KUKA KRL program: EPS_2_25252_SD1A_A_20250910061717.src

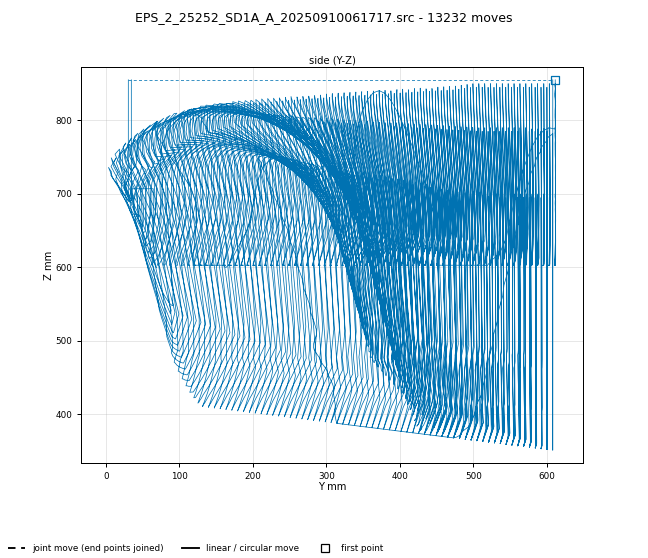
[picture p0: tool path of EPS_2_25252_SD1A_A_20250910061717.src, 13232 of 13234 moves have a stored position in this frame; points joined in program order, loops and branches not executed]
&ACCESS RVP
&REL 4
&COMMENT QRS 19112012
&PARAM EDITMASK = *
DEF PART()
EXT BAS (BAS_COMMAND :IN,REAL :IN )
INT I
BAS (#INITMOV,0 )

;KUKA QRS Post kuka4.cps  Date:22-06-2017 !

File_ID=2822

QRS_PRE_INIT()

;Init var - Until changes are made in qrs_pre_init
Outlet_Square_prg=0
Inlet_1_Square_prg=0
Inlet_2_Square_prg=0
Inlet_3_Square_prg=0
Inlet_4_Square_prg=0
Inlet_5_Square_prg=0

Outlet_1={X 0.000, Y 501.250, Z 662.000, B 0.000, E1 0.000 }
Inlet_1={X 0.000, Y 505.750, Z 602.000, B 0.000, E1 90.000 }
Inlet_2={X 0.000, Y 531.500, Z 514.500, B 0.000, E1 270.000 }
Outlet_1_type=366
Inlet_1_type=366
Inlet_2_type=201
;QRS#1=Sidecore dimensions
;QRS#2=375-15" PVC SDR 35
;QRS#3=375-15" PVC SDR 35
;QRS#4=200-8" PVC SDR 35
;QRS#5=
;QRS#6=
;QRS#7=
;QRS#8=
;QRS#9=20Y PSX
;QRS#10=20Y PSX
;QRS#11=12-08 PSX
;QRS#12=
;QRS#13=
;QRS#14=
;QRS#15=
;QRS#16=1220x127x1143 3,75'
;QRS#17=EPS Height
;QRS#18=845
;QRS#19=*
;QRS#20= UPDATED VERSION 22-06-2017
;QRS#21=*
Outlet_Square=0250
Inlet_1_Square=0250
Inlet_2_Square=0100
Inlet_3_Square=0
Inlet_4_Square=0
Inlet_5_Square=0
Mill_Square=1
Outlet_Square_Prg=252
Inlet_1_Square_prg=252
Inlet_2_Square_prg=204

QRS_INIT()

$ADVANCE=5

; T1
PTP {E1 176.989,E2 176.989}
PTP {X 0,Y 611.255,A -85,B 0,C 180,E1 176.989,E2 176.989,E3 0,E4 0,E5 0,E6 0}
QRS_SPEED_INIT()
LIN {X 0,Y 611.255,Z 855,A -85,B 0,C 180,E1 176.989,E2 176.989,E3 0,E4 0,E5 0,E6 0} C_VEL
LIN {X 0,Y 611.255,Z 797.706,A -85,B 0,C 180,E1 176.989,E2 176.989} C_VEL
LIN {X 0,Y 611.255,Z 789.909,A -85,B 0,C 180,E1 176.989,E2 176.989} C_VEL
LIN {X 0,Y 611.338,Z 787.921,A -85,B 0,C 180,E1 177.197,E2 177.197} C_VEL
LIN {X 0,Y 611.834,Z 789.089,A -85,B 0,C 180,E1 178.169,E2 178.169} C_VEL
LIN {X 0,Y 611.558,Z 789.587,A -85,B 0,C 180,E1 178.832,E2 178.832} C_VEL
LIN {X 0,Y 611.055,Z 789.944,A -85,B 0,C 180,E1 179.766,E2 179.766} C_VEL
LIN {X 0,Y 610.786,Z 789.821,A -85,B 0,C 180,E1 180.701,E2 180.701} C_VEL
LIN {X 0,Y 610.813,Z 789.552,A -85,B 0,C 180,E1 181.169,E2 181.169} C_VEL
LIN {X 0,Y 611.351,Z 788.136,A -85,B 0,C 180,E1 182.57,E2 182.57} C_VEL
LIN {X 0,Y 611.881,Z 786.565,A -85,B 0,C 180,E1 183.503,E2 183.503} C_VEL
LIN {X 0,Y 611.302,Z 783.918,A -85,B 0,C 180,E1 184.677,E2 184.677} C_VEL
LIN {X 0,Y 611.043,Z 782.348,A -85,B 0,C 180,E1 185.266,E2 185.266} C_VEL
LIN {X 0,Y 610.913,Z 779.545,A -85,B 0,C 180,E1 186.148,E2 186.148} C_VEL
LIN {X 0,Y 611.141,Z 776.265,A -85,B 0,C 180,E1 187.027,E2 187.027} C_VEL
LIN {X 0,Y 611.585,Z 772.483,A -85,B 0,C 180,E1 187.905,E2 187.905} C_VEL
LIN {X 0,Y 611.869,Z 769.622,A -85,B 0,C 180,E1 188.491,E2 188.491} C_VEL
LIN {X 0,Y 611.527,Z 764.94,A -85,B 0,C 180,E1 189.382,E2 189.382} C_VEL
LIN {X 0,Y 611.202,Z 759.672,A -85,B 0,C 180,E1 190.276,E2 190.276} C_VEL
LIN {X 0,Y 611.223,Z 752.664,A -85,B 0,C 180,E1 191.317,E2 191.317} C_VEL
LIN {X 0,Y 611.512,Z 747.064,A -85,B 0,C 180,E1 192.056,E2 192.056} C_VEL
LIN {X 0,Y 611.803,Z 740.897,A -85,B 0,C 180,E1 192.797,E2 192.797} C_VEL
LIN {X 0,Y 611.777,Z 735.91,A -85,B 0,C 180,E1 193.359,E2 193.359} C_VEL
LIN {X 0,Y 611.519,Z 727.994,A -85,B 0,C 180,E1 194.172,E2 194.172} C_VEL
LIN {X 0,Y 611.4,Z 721.632,A -85,B 0,C 180,E1 194.769,E2 194.769} C_VEL
LIN {X 0,Y 611.46,Z 714.699,A -85,B 0,C 180,E1 195.363,E2 195.363} C_VEL
LIN {X 0,Y 611.677,Z 706.786,A -85,B 0,C 180,E1 195.978,E2 195.978} C_VEL
LIN {X 0,Y 611.783,Z 698.644,A -85,B 0,C 180,E1 196.557,E2 196.557} C_VEL
LIN {X 0,Y 611.811,Z 690.326,A -85,B 0,C 180,E1 197.094,E2 197.094} C_VEL
LIN {X 0,Y 611.741,Z 682.443,A -85,B 0,C 180,E1 197.56,E2 197.56} C_VEL
LIN {X 0,Y 611.722,Z 675.291,A -85,B 0,C 180,E1 197.945,E2 197.945} C_VEL
LIN {X 0,Y 611.776,Z 665.714,A -85,B 0,C 180,E1 198.404,E2 198.404} C_VEL
LIN {X 0,Y 611.781,Z 656.669,A -85,B 0,C 180,E1 198.789,E2 198.789} C_VEL
LIN {X 0,Y 611.797,Z 648.504,A -85,B 0,C 180,E1 199.097,E2 199.097} C_VEL
LIN {X 0,Y 611.848,Z 637.724,A -85,B 0,C 180,E1 199.443,E2 199.443} C_VEL
LIN {X 0,Y 611.821,Z 629.276,A -85,B 0,C 180,E1 199.676,E2 199.676} C_VEL
LIN {X 0,Y 611.827,Z 618.943,A -85,B 0,C 180,E1 199.908,E2 199.908} C_VEL
LIN {X 0,Y 611.776,Z 610.345,A -85,B 0,C 180,E1 200.065,E2 200.065} C_VEL
LIN {X 0,Y 611.596,Z 602.81,A -85,B 0,C 180,E1 200.188,E2 200.188} C_VEL
LIN {X 0,Y 611.78,Z 602.81,A -85,B 0,C 180,E1 200.26,E2 200.26} C_VEL
LIN {X 0,Y 611.752,Z 602.81,A -85,B 0,C 180,E1 207.938,E2 207.938} C_VEL
LIN {X 0,Y 610.419,Z 602.81,A -85,B 0,C 180,E1 210.688,E2 210.688} C_VEL
LIN {X 0,Y 611.718,Z 602.81,A -85,B 0,C 180,E1 216.211,E2 216.211} C_VEL
LIN {X 0,Y 611.159,Z 602.81,A -85,B 0,C 180,E1 217.326,E2 217.326} C_VEL
LIN {X 0,Y 610.678,Z 602.81,A -85,B 0,C 180,E1 222.329,E2 222.329} C_VEL
LIN {X 0,Y 611.693,Z 602.81,A -85,B 0,C 180,E1 224.519,E2 224.519} C_VEL
LIN {X 0,Y 611.666,Z 602.81,A -85,B 0,C 180,E1 232.612,E2 232.612} C_VEL
LIN {X 0,Y 611.151,Z 602.81,A -85,B 0,C 180,E1 233.75,E2 233.75} C_VEL
LIN {X 0,Y 611.656,Z 602.81,A -85,B 0,C 180,E1 241.169,E2 241.169} C_VEL
LIN {X 0,Y 611.476,Z 602.81,A -85,B 0,C 180,E1 242.049,E2 242.049} C_VEL
LIN {X 0,Y 611.803,Z 602.81,A -85,B 0,C 180,E1 248.625,E2 248.625} C_VEL
LIN {X 0,Y 610.997,Z 602.81,A -85,B 0,C 180,E1 248.983,E2 248.983} C_VEL
LIN {X 0,Y 610.769,Z 602.853,A -85,B 0,C 180,E1 249.009,E2 249.009} C_VEL
LIN {X 0,Y 611.62,Z 640.893,A -85,B 0,C 180,E1 249.507,E2 249.507} C_VEL
LIN {X 0,Y 611.825,Z 668.068,A -85,B 0,C 180,E1 249.859,E2 249.859} C_VEL
LIN {X 0,Y 611.844,Z 677.232,A -85,B 0,C 180,E1 250.014,E2 250.014} C_VEL
LIN {X 0,Y 611.82,Z 686.284,A -85,B 0,C 180,E1 250.208,E2 250.208} C_VEL
LIN {X 0,Y 611.674,Z 695.239,A -85,B 0,C 180,E1 250.435,E2 250.435} C_VEL
LIN {X 0,Y 611.805,Z 704.1,A -85,B 0,C 180,E1 250.71,E2 250.71} C_VEL
LIN {X 0,Y 611.808,Z 711.864,A -85,B 0,C 180,E1 250.981,E2 250.981} C_VEL
LIN {X 0,Y 611.808,Z 721.496,A -85,B 0,C 180,E1 251.366,E2 251.366} C_VEL
LIN {X 0,Y 611.827,Z 729.998,A -85,B 0,C 180,E1 251.751,E2 251.751} C_VEL
LIN {X 0,Y 611.756,Z 739.053,A -85,B 0,C 180,E1 252.209,E2 252.209} C_VEL
LIN {X 0,Y 611.731,Z 748.469,A -85,B 0,C 180,E1 252.745,E2 252.745} C_VEL
LIN {X 0,Y 611.565,Z 756.855,A -85,B 0,C 180,E1 253.272,E2 253.272} C_VEL
LIN {X 0,Y 611.462,Z 763.316,A -85,B 0,C 180,E1 253.715,E2 253.715} C_VEL
LIN {X 0,Y 611.523,Z 770.776,A -85,B 0,C 180,E1 254.277,E2 254.277} C_VEL
LIN {X 0,Y 611.733,Z 778.696,A -85,B 0,C 180,E1 254.937,E2 254.937} C_VEL
LIN {X 0,Y 611.827,Z 785.197,A -85,B 0,C 180,E1 255.523,E2 255.523} C_VEL
LIN {X 0,Y 611.641,Z 792.111,A -85,B 0,C 180,E1 256.198,E2 256.198} C_VEL
LIN {X 0,Y 611.381,Z 798.097,A -85,B 0,C 180,E1 256.831,E2 256.831} C_VEL
LIN {X 0,Y 611.254,Z 803.807,A -85,B 0,C 180,E1 257.49,E2 257.49} C_VEL
LIN {X 0,Y 611.36,Z 809.701,A -85,B 0,C 180,E1 258.239,E2 258.239} C_VEL
LIN {X 0,Y 611.556,Z 814.069,A -85,B 0,C 180,E1 258.838,E2 258.838} C_VEL
LIN {X 0,Y 611.862,Z 819.944,A -85,B 0,C 180,E1 259.735,E2 259.735} C_VEL
LIN {X 0,Y 611.48,Z 825.185,A -85,B 0,C 180,E1 260.617,E2 260.617} C_VEL
LIN {X 0,Y 611.206,Z 828.398,A -85,B 0,C 180,E1 261.204,E2 261.204} C_VEL
LIN {X 0,Y 611.051,Z 832.684,A -85,B 0,C 180,E1 262.088,E2 262.088} C_VEL
LIN {X 0,Y 611.215,Z 836.436,A -85,B 0,C 180,E1 262.974,E2 262.974} C_VEL
LIN {X 0,Y 611.602,Z 839.681,A -85,B 0,C 180,E1 263.859,E2 263.859} C_VEL
LIN {X 0,Y 611.753,Z 840.616,A -85,B 0,C 180,E1 264.154,E2 264.154} C_VEL
LIN {X 0,Y 611.721,Z 842.453,A -85,B 0,C 180,E1 264.74,E2 264.74} C_VEL
LIN {X 0,Y 611.158,Z 845.43,A -85,B 0,C 180,E1 265.908,E2 265.908} C_VEL
LIN {X 0,Y 610.966,Z 846.682,A -85,B 0,C 180,E1 266.492,E2 266.492} C_VEL
LIN {X 0,Y 611.091,Z 848.544,A -85,B 0,C 180,E1 267.72,E2 267.72} C_VEL
LIN {X 0,Y 611.598,Z 849.552,A -85,B 0,C 180,E1 268.833,E2 268.833} C_VEL
LIN {X 0,Y 611.713,Z 849.903,A -85,B 0,C 180,E1 269.767,E2 269.767} C_VEL
LIN {X 0,Y 611.245,Z 849.816,A -85,B 0,C 180,E1 270.701,E2 270.701} C_VEL
LIN {X 0,Y 610.955,Z 848.959,A -85,B 0,C 180,E1 271.933,E2 271.933} C_VEL
LIN {X 0,Y 611.441,Z 846.667,A -85,B 0,C 180,E1 273.505,E2 273.505} C_VEL
LIN {X 0,Y 611.736,Z 845.409,A -85,B 0,C 180,E1 274.088,E2 274.088} C_VEL
LIN {X 0,Y 611.745,Z 844.023,A -85,B 0,C 180,E1 274.674,E2 274.674} C_VEL
LIN {X 0,Y 611.452,Z 842.462,A -85,B 0,C 180,E1 275.262,E2 275.262} C_VEL
LIN {X 0,Y 611.033,Z 839.69,A -85,B 0,C 180,E1 276.146,E2 276.146} C_VEL
LIN {X 0,Y 610.903,Z 836.436,A -85,B 0,C 180,E1 277.03,E2 277.03} C_VEL
LIN {X 0,Y 611.133,Z 832.684,A -85,B 0,C 180,E1 277.911,E2 277.911} C_VEL
LIN {X 0,Y 611.587,Z 828.398,A -85,B 0,C 180,E1 278.79,E2 278.79} C_VEL
LIN {X 0,Y 611.871,Z 825.185,A -85,B 0,C 180,E1 279.377,E2 279.377} C_VEL
LIN {X 0,Y 611.518,Z 819.944,A -85,B 0,C 180,E1 280.271,E2 280.271} C_VEL
LIN {X 0,Y 611.154,Z 812.996,A -85,B 0,C 180,E1 281.318,E2 281.318} C_VEL
LIN {X 0,Y 611.164,Z 807.427,A -85,B 0,C 180,E1 282.063,E2 282.063} C_VEL
LIN {X 0,Y 611.414,Z 801.293,A -85,B 0,C 180,E1 282.806,E2 282.806} C_VEL
LIN {X 0,Y 611.786,Z 793.803,A -85,B 0,C 180,E1 283.623,E2 283.623} C_VEL
LIN {X 0,Y 611.787,Z 787.856,A -85,B 0,C 180,E1 284.223,E2 284.223} C_VEL
LIN {X 0,Y 611.566,Z 780.74,A -85,B 0,C 180,E1 284.888,E2 284.888} C_VEL
LIN {X 0,Y 611.417,Z 774.124,A -85,B 0,C 180,E1 285.456,E2 285.456} C_VEL
LIN {X 0,Y 611.438,Z 767.139,A -85,B 0,C 180,E1 286.004,E2 286.004} C_VEL
LIN {X 0,Y 611.599,Z 759.502,A -85,B 0,C 180,E1 286.549,E2 286.549} C_VEL
LIN {X 0,Y 611.777,Z 751.324,A -85,B 0,C 180,E1 287.079,E2 287.079} C_VEL
LIN {X 0,Y 611.815,Z 743.302,A -85,B 0,C 180,E1 287.555,E2 287.555} C_VEL
LIN {X 0,Y 611.798,Z 734.646,A -85,B 0,C 180,E1 288.02,E2 288.02} C_VEL
LIN {X 0,Y 611.708,Z 726.729,A -85,B 0,C 180,E1 288.407,E2 288.407} C_VEL
LIN {X 0,Y 611.712,Z 717.825,A -85,B 0,C 180,E1 288.791,E2 288.791} C_VEL
LIN {X 0,Y 611.801,Z 707.539,A -85,B 0,C 180,E1 289.174,E2 289.174} C_VEL
LIN {X 0,Y 611.768,Z 697.93,A -85,B 0,C 180,E1 289.484,E2 289.484} C_VEL
LIN {X 0,Y 611.774,Z 691.134,A -85,B 0,C 180,E1 289.678,E2 289.678} C_VEL
LIN {X 0,Y 611.852,Z 679.255,A -85,B 0,C 180,E1 289.946,E2 289.946} C_VEL
LIN {X 0,Y 611.842,Z 669.403,A -85,B 0,C 180,E1 290.121,E2 290.121} C_VEL
LIN {X 0,Y 611.69,Z 646.222,A -85,B 0,C 180,E1 290.425,E2 290.425} C_VEL
LIN {X 0,Y 610.919,Z 608.013,A -85,B 0,C 180,E1 290.922,E2 290.922} C_VEL
LIN {X 0,Y 610.821,Z 602.81,A -85,B 0,C 180,E1 290.998,E2 290.998} C_VEL
LIN {X 0,Y 611.662,Z 602.81,A -85,B 0,C 180,E1 291.131,E2 291.131} C_VEL
LIN {X 0,Y 611.599,Z 602.81,A -85,B 0,C 180,E1 291.733,E2 291.733} C_VEL
LIN {X 0,Y 611.815,Z 602.81,A -85,B 0,C 180,E1 297.934,E2 297.934} C_VEL
LIN {X 0,Y 610.481,Z 602.81,A -85,B 0,C 180,E1 300.684,E2 300.684} C_VEL
LIN {X 0,Y 611.803,Z 602.81,A -85,B 0,C 180,E1 306.205,E2 306.205} C_VEL
LIN {X 0,Y 611.22,Z 602.81,A -85,B 0,C 180,E1 307.333,E2 307.333} C_VEL
LIN {X 0,Y 610.732,Z 602.81,A -85,B 0,C 180,E1 312.325,E2 312.325} C_VEL
LIN {X 0,Y 611.759,Z 602.81,A -85,B 0,C 180,E1 314.525,E2 314.525} C_VEL
LIN {X 0,Y 611.719,Z 602.81,A -85,B 0,C 180,E1 322.605,E2 322.605} C_VEL
LIN {X 0,Y 611.181,Z 602.81,A -85,B 0,C 180,E1 323.752,E2 323.752} C_VEL
LIN {X 0,Y 611.606,Z 602.81,A -85,B 0,C 180,E1 331.178,E2 331.178} C_VEL
LIN {X 0,Y 611.391,Z 602.81,A -85,B 0,C 180,E1 332.044,E2 332.044} C_VEL
LIN {X 0,Y 611.822,Z 602.81,A -85,B 0,C 180,E1 339.742,E2 339.742} C_VEL
LIN {X 0,Y 611.83,Z 602.81,A -85,B 0,C 180,E1 347.842,E2 347.842} C_VEL
LIN {X 0,Y 611.645,Z 602.89,A -85,B 0,C 180,E1 348.052,E2 348.052} C_VEL
LIN {X 0,Y 611.831,Z 610.86,A -85,B 0,C 180,E1 348.286,E2 348.286} C_VEL
LIN {X 0,Y 611.839,Z 619.207,A -85,B 0,C 180,E1 348.582,E2 348.582} C_VEL
LIN {X 0,Y 611.857,Z 627.631,A -85,B 0,C 180,E1 348.949,E2 348.949} C_VEL
LIN {X 0,Y 611.843,Z 635.937,A -85,B 0,C 180,E1 349.377,E2 349.377} C_VEL
LIN {X 0,Y 611.694,Z 643.024,A -85,B 0,C 180,E1 349.806,E2 349.806} C_VEL
LIN {X 0,Y 611.601,Z 650.478,A -85,B 0,C 180,E1 350.323,E2 350.323} C_VEL
LIN {X 0,Y 611.746,Z 657.755,A -85,B 0,C 180,E1 350.917,E2 350.917} C_VEL
LIN {X 0,Y 611.865,Z 664.105,A -85,B 0,C 180,E1 351.509,E2 351.509} C_VEL
LIN {X 0,Y 611.633,Z 669.644,A -85,B 0,C 180,E1 352.095,E2 352.095} C_VEL
LIN {X 0,Y 611.278,Z 675.666,A -85,B 0,C 180,E1 352.827,E2 352.827} C_VEL
LIN {X 0,Y 611.236,Z 678.856,A -85,B 0,C 180,E1 353.268,E2 353.268} C_VEL
LIN {X 0,Y 611.382,Z 682.66,A -85,B 0,C 180,E1 353.857,E2 353.857} C_VEL
LIN {X 0,Y 611.667,Z 686.017,A -85,B 0,C 180,E1 354.447,E2 354.447} C_VEL
LIN {X 0,Y 611.88,Z 688.956,A -85,B 0,C 180,E1 355.035,E2 355.035} C_VEL
LIN {X 0,Y 611.599,Z 691.514,A -85,B 0,C 180,E1 355.618,E2 355.618} C_VEL
LIN {X 0,Y 611.128,Z 694.638,A -85,B 0,C 180,E1 356.493,E2 356.493} C_VEL
LIN {X 0,Y 611.022,Z 696.481,A -85,B 0,C 180,E1 357.14,E2 357.14} C_VEL
LIN {X 0,Y 611.323,Z 698.328,A -85,B 0,C 180,E1 358.032,E2 358.032} C_VEL
LIN {X 0,Y 611.76,Z 699.395,A -85,B 0,C 180,E1 358.833,E2 358.833} C_VEL
LIN {X 0,Y 611.815,Z 699.742,A -85,B 0,C 180,E1 359.3,E2 359.3} C_VEL
LIN {X 0,Y 611.316,Z 699.913,A -85,B 0,C 180,E1 360.234,E2 360.234} C_VEL
LIN {X 0,Y 611.123,Z 699.712,A -85,B 0,C 180,E1 360.701,E2 360.701} C_VEL
LIN {X 0,Y 611.058,Z 699.321,A -85,B 0,C 180,E1 361.169,E2 361.169} C_VEL
LIN {X 0,Y 611.126,Z 698.739,A -85,B 0,C 180,E1 361.636,E2 361.636} C_VEL
LIN {X 0,Y 611.568,Z 696.941,A -85,B 0,C 180,E1 362.569,E2 362.569} C_VEL
LIN {X 0,Y 611.798,Z 695.73,A -85,B 0,C 180,E1 363.036,E2 363.036} C_VEL
LIN {X 0,Y 611.681,Z 693.755,A -85,B 0,C 180,E1 363.684,E2 363.684} C_VEL
LIN {X 0,Y 611.326,Z 691.141,A -85,B 0,C 180,E1 364.384,E2 364.384} C_VEL
LIN {X 0,Y 611.126,Z 687.101,A -85,B 0,C 180,E1 365.265,E2 365.265} C_VEL
LIN {X 0,Y 611.288,Z 683.901,A -85,B 0,C 180,E1 365.85,E2 365.85} C_VEL
LIN {X 0,Y 611.771,Z 678.248,A -85,B 0,C 180,E1 366.726,E2 366.726} C_VEL
LIN {X 0,Y 611.814,Z 673.838,A -85,B 0,C 180,E1 367.314,E2 367.314} C_VEL
LIN {X 0,Y 611.505,Z 667.518,A -85,B 0,C 180,E1 368.054,E2 368.054} C_VEL
LIN {X 0,Y 611.396,Z 661.645,A -85,B 0,C 180,E1 368.645,E2 368.645} C_VEL
LIN {X 0,Y 611.567,Z 654.978,A -85,B 0,C 180,E1 369.234,E2 369.234} C_VEL
LIN {X 0,Y 611.802,Z 647.181,A -85,B 0,C 180,E1 369.822,E2 369.822} C_VEL
LIN {X 0,Y 611.792,Z 639.219,A -85,B 0,C 180,E1 370.341,E2 370.341} C_VEL
LIN {X 0,Y 611.673,Z 631.524,A -85,B 0,C 180,E1 370.773,E2 370.773} C_VEL
LIN {X 0,Y 611.667,Z 624.263,A -85,B 0,C 180,E1 371.119,E2 371.119} C_VEL
LIN {X 0,Y 611.771,Z 615.833,A -85,B 0,C 180,E1 371.456,E2 371.456} C_VEL
LIN {X 0,Y 611.596,Z 606.761,A -85,B 0,C 180,E1 371.753,E2 371.753} C_VEL
LIN {X 0,Y 611.3,Z 602.81,A -85,B 0,C 180,E1 371.869,E2 371.869} C_VEL
LIN {X 0,Y 611.817,Z 602.81,A -85,B 0,C 180,E1 372.031,E2 372.031} C_VEL
LIN {X 0,Y 611.863,Z 602.81,A -85,B 0,C 180,E1 375.353,E2 375.353} C_VEL
LIN {X 0,Y 611.809,Z 602.81,A -85,B 0,C 180,E1 382.768,E2 382.768} C_VEL
LIN {X 0,Y 611.758,Z 602.81,A -85,B 0,C 180,E1 390.614,E2 390.614} C_VEL
LIN {X 0,Y 611.738,Z 602.81,A -85,B 0,C 180,E1 399.16,E2 399.16} C_VEL
LIN {X 0,Y 610.339,Z 602.81,A -85,B 0,C 180,E1 402.358,E2 402.358} C_VEL
LIN {X 0,Y 610.662,Z 602.81,A -85,B 0,C 180,E1 405.579,E2 405.579} C_VEL
LIN {X 0,Y 611.756,Z 602.81,A -85,B 0,C 180,E1 407.763,E2 407.763} C_VEL
LIN {X 0,Y 610.231,Z 602.81,A -85,B 0,C 180,E1 413.687,E2 413.687} C_VEL
LIN {X 0,Y 611.725,Z 602.81,A -85,B 0,C 180,E1 416.637,E2 416.637} C_VEL
LIN {X 0,Y 611.755,Z 602.81,A -85,B 0,C 180,E1 424.674,E2 424.674} C_VEL
LIN {X 0,Y 611.535,Z 602.81,A -85,B 0,C 180,E1 433.281,E2 433.281} C_VEL
LIN {X 0,Y 611.288,Z 602.81,A -85,B 0,C 180,E1 434.632,E2 434.632} C_VEL
LIN {X 0,Y 611.867,Z 602.81,A -85,B 0,C 180,E1 441.804,E2 441.804} C_VEL
LIN {X 0,Y 611.811,Z 602.81,A -85,B 0,C 180,E1 448.833,E2 448.833} C_VEL
LIN {X 0,Y 611.843,Z 602.81,A -85,B 0,C 180,E1 455.845,E2 455.845} C_VEL
LIN {X 0,Y 611.779,Z 602.81,A -85,B 0,C 180,E1 462.948,E2 462.948} C_VEL
LIN {X 0,Y 611.839,Z 602.81,A -85,B 0,C 180,E1 470.258,E2 470.258} C_VEL
LIN {X 0,Y 611.8,Z 602.81,A -85,B 0,C 180,E1 477.935,E2 477.935} C_VEL
LIN {X 0,Y 610.463,Z 602.81,A -85,B 0,C 180,E1 480.685,E2 480.685} C_VEL
LIN {X 0,Y 611.789,Z 602.81,A -85,B 0,C 180,E1 486.206,E2 486.206} C_VEL
LIN {X 0,Y 611.218,Z 602.81,A -85,B 0,C 180,E1 487.333,E2 487.333} C_VEL
LIN {X 0,Y 610.726,Z 602.81,A -85,B 0,C 180,E1 492.325,E2 492.325} C_VEL
LIN {X 0,Y 611.752,Z 602.81,A -85,B 0,C 180,E1 494.525,E2 494.525} C_VEL
LIN {X 0,Y 611.716,Z 602.81,A -85,B 0,C 180,E1 502.606,E2 502.606} C_VEL
LIN {X 0,Y 611.188,Z 602.81,A -85,B 0,C 180,E1 503.752,E2 503.752} C_VEL
LIN {X 0,Y 611.615,Z 602.81,A -85,B 0,C 180,E1 511.176,E2 511.176} C_VEL
LIN {X 0,Y 611.407,Z 602.81,A -85,B 0,C 180,E1 512.045,E2 512.045} C_VEL
LIN {X 0,Y 611.692,Z 602.81,A -85,B 0,C 180,E1 519.149,E2 519.149} C_VEL
LIN {X 0,Y 611.768,Z 602.81,A -85,B 0,C 180,E1 519.446,E2 519.446} C_VEL
LIN {X 0,Y 611.265,Z 602.81,A -85,B 0,C 180,E1 519.576,E2 519.576} C_VEL
LIN {X 0,Y 610.267,Z 602.828,A -85,B 0,C 180,E1 519.685,E2 519.685} C_VEL
LIN {X 0,Y 611.272,Z 612.441,A -85,B 0,C 180,E1 519.859,E2 519.859} C_VEL
LIN {X 0,Y 611.669,Z 623.322,A -85,B 0,C 180,E1 520.086,E2 520.086} C_VEL
LIN {X 0,Y 611.784,Z 634.126,A -85,B 0,C 180,E1 520.361,E2 520.361} C_VEL
LIN {X 0,Y 611.789,Z 644.296,A -85,B 0,C 180,E1 520.671,E2 520.671} C_VEL
LIN {X 0,Y 611.736,Z 653.028,A -85,B 0,C 180,E1 520.978,E2 520.978} C_VEL
LIN {X 0,Y 611.795,Z 662.522,A -85,B 0,C 180,E1 521.365,E2 521.365} C_VEL
LIN {X 0,Y 611.686,Z 670.911,A -85,B 0,C 180,E1 521.746,E2 521.746} C_VEL
LIN {X 0,Y 611.578,Z 678.481,A -85,B 0,C 180,E1 522.127,E2 522.127} C_VEL
LIN {X 0,Y 611.6,Z 686.735,A -85,B 0,C 180,E1 522.59,E2 522.59} C_VEL
LIN {X 0,Y 611.762,Z 695.828,A -85,B 0,C 180,E1 523.163,E2 523.163} C_VEL
LIN {X 0,Y 611.799,Z 703.879,A -85,B 0,C 180,E1 523.72,E2 523.72} C_VEL
LIN {X 0,Y 611.792,Z 711.228,A -85,B 0,C 180,E1 524.276,E2 524.276} C_VEL
LIN {X 0,Y 611.759,Z 719.348,A -85,B 0,C 180,E1 524.95,E2 524.95} C_VEL
LIN {X 0,Y 611.571,Z 726.055,A -85,B 0,C 180,E1 525.554,E2 525.554} C_VEL
LIN {X 0,Y 611.413,Z 731.236,A -85,B 0,C 180,E1 526.056,E2 526.056} C_VEL
LIN {X 0,Y 611.386,Z 738.639,A -85,B 0,C 180,E1 526.848,E2 526.848} C_VEL
LIN {X 0,Y 611.598,Z 745.378,A -85,B 0,C 180,E1 527.647,E2 527.647} C_VEL
LIN {X 0,Y 611.828,Z 751.131,A -85,B 0,C 180,E1 528.397,E2 528.397} C_VEL
LIN {X 0,Y 611.749,Z 754.371,A -85,B 0,C 180,E1 528.842,E2 528.842} C_VEL
LIN {X 0,Y 611.327,Z 760.216,A -85,B 0,C 180,E1 529.726,E2 529.726} C_VEL
LIN {X 0,Y 611.106,Z 763.803,A -85,B 0,C 180,E1 530.315,E2 530.315} C_VEL
LIN {X 0,Y 611.059,Z 768.625,A -85,B 0,C 180,E1 531.202,E2 531.202} C_VEL
LIN {X 0,Y 611.34,Z 772.878,A -85,B 0,C 180,E1 532.092,E2 532.092} C_VEL
LIN {X 0,Y 611.775,Z 776.597,A -85,B 0,C 180,E1 532.98,E2 532.98} C_VEL
LIN {X 0,Y 611.878,Z 777.692,A -85,B 0,C 180,E1 533.275,E2 533.275} C_VEL
LIN {X 0,Y 611.442,Z 780.768,A -85,B 0,C 180,E1 534.151,E2 534.151} C_VEL
LIN {X 0,Y 611.145,Z 782.59,A -85,B 0,C 180,E1 534.735,E2 534.735} C_VEL
LIN {X 0,Y 610.968,Z 784.166,A -85,B 0,C 180,E1 535.32,E2 535.32} C_VEL
LIN {X 0,Y 611.045,Z 786.755,A -85,B 0,C 180,E1 536.492,E2 536.492} C_VEL
LIN {X 0,Y 611.338,Z 787.921,A -85,B 0,C 180,E1 537.197,E2 537.197} C_VEL
LIN {X 0,Y 602.858,Z 789.832,A -85,B 0,C 180,E1 540.462,E2 540.462} C_VEL
LIN {X 0,Y 603.127,Z 783.101,A -85,B 0,C 180,E1 545.053,E2 545.053} C_VEL
LIN {X 0,Y 603.366,Z 762.386,A -85,B 0,C 180,E1 549.958,E2 549.958} C_VEL
LIN {X 0,Y 603.623,Z 727.935,A -85,B 0,C 180,E1 554.368,E2 554.368} C_VEL
LIN {X 0,Y 604.042,Z 681.758,A -85,B 0,C 180,E1 557.83,E2 557.83} C_VEL
LIN {X 0,Y 604.275,Z 629.84,A -85,B 0,C 180,E1 559.92,E2 559.92} C_VEL
LIN {X 0,Y 603.494,Z 602.81,A -85,B 0,C 180,E1 560.659,E2 560.659} C_VEL
LIN {X 0,Y 602.733,Z 602.81,A -85,B 0,C 180,E1 569.736,E2 569.736} C_VEL
LIN {X 0,Y 603.037,Z 602.81,A -85,B 0,C 180,E1 577.59,E2 577.59} C_VEL
LIN {X 0,Y 602.697,Z 602.81,A -85,B 0,C 180,E1 586.2,E2 586.2} C_VEL
LIN {X 0,Y 603.125,Z 602.81,A -85,B 0,C 180,E1 593.771,E2 593.771} C_VEL
LIN {X 0,Y 602.929,Z 602.81,A -85,B 0,C 180,E1 603.316,E2 603.316} C_VEL
LIN {X 0,Y 603.375,Z 602.81,A -85,B 0,C 180,E1 608.724,E2 608.724} C_VEL
LIN {X 0,Y 604.141,Z 697.306,A -85,B 0,C 180,E1 610.241,E2 610.241} C_VEL
LIN {X 0,Y 604.015,Z 749.181,A -85,B 0,C 180,E1 612.562,E2 612.562} C_VEL
LIN {X 0,Y 603.805,Z 792.189,A -85,B 0,C 180,E1 616.023,E2 616.023} C_VEL
LIN {X 0,Y 603.489,Z 825.8,A -85,B 0,C 180,E1 620.606,E2 620.606} C_VEL
LIN {X 0,Y 603.258,Z 845.076,A -85,B 0,C 180,E1 625.684,E2 625.684} C_VEL
LIN {X 0,Y 603.246,Z 849.836,A -85,B 0,C 180,E1 630.732,E2 630.732} C_VEL
LIN {X 0,Y 603.196,Z 841.081,A -85,B 0,C 180,E1 635.787,E2 635.787} C_VEL
LIN {X 0,Y 603.408,Z 818.13,A -85,B 0,C 180,E1 640.7,E2 640.7} C_VEL
LIN {X 0,Y 603.723,Z 782.041,A -85,B 0,C 180,E1 644.97,E2 644.97} C_VEL
LIN {X 0,Y 604.125,Z 735.468,A -85,B 0,C 180,E1 648.216,E2 648.216} C_VEL
LIN {X 0,Y 604.336,Z 683.617,A -85,B 0,C 180,E1 650.113,E2 650.113} C_VEL
LIN {X 0,Y 603.648,Z 602.81,A -85,B 0,C 180,E1 651.388,E2 651.388} C_VEL
LIN {X 0,Y 602.799,Z 602.81,A -85,B 0,C 180,E1 659.713,E2 659.713} C_VEL
LIN {X 0,Y 603.087,Z 602.81,A -85,B 0,C 180,E1 667.569,E2 667.569} C_VEL
LIN {X 0,Y 602.773,Z 602.81,A -85,B 0,C 180,E1 676.185,E2 676.185} C_VEL
LIN {X 0,Y 603.18,Z 602.81,A -85,B 0,C 180,E1 683.756,E2 683.756} C_VEL
LIN {X 0,Y 603.244,Z 602.81,A -85,B 0,C 180,E1 692.264,E2 692.264} C_VEL
LIN {X 0,Y 602.727,Z 602.81,A -85,B 0,C 180,E1 701.655,E2 701.655} C_VEL
LIN {X 0,Y 603.838,Z 604.542,A -85,B 0,C 180,E1 707.941,E2 707.941} C_VEL
LIN {X 0,Y 603.794,Z 644.574,A -85,B 0,C 180,E1 709.775,E2 709.775} C_VEL
LIN {X 0,Y 603.305,Z 675.973,A -85,B 0,C 180,E1 712.774,E2 712.774} C_VEL
LIN {X 0,Y 603.171,Z 694.47,A -85,B 0,C 180,E1 716.393,E2 716.393} C_VEL
LIN {X 0,Y 603.839,Z 699.789,A -85,B 0,C 180,E1 719.279,E2 719.279} C_VEL
LIN {X 0,Y 603.719,Z 694.193,A -85,B 0,C 180,E1 723.602,E2 723.602} C_VEL
LIN {X 0,Y 603.841,Z 674.312,A -85,B 0,C 180,E1 727.351,E2 727.351} C_VEL
LIN {X 0,Y 603.906,Z 641.868,A -85,B 0,C 180,E1 730.312,E2 730.312} C_VEL
LIN {X 0,Y 603.786,Z 602.81,A -85,B 0,C 180,E1 732.15,E2 732.15} C_VEL
LIN {X 0,Y 602.641,Z 602.81,A -85,B 0,C 180,E1 739.872,E2 739.872} C_VEL
LIN {X 0,Y 602.801,Z 602.81,A -85,B 0,C 180,E1 744.541,E2 744.541} C_VEL
LIN {X 0,Y 602.596,Z 602.81,A -85,B 0,C 180,E1 752.462,E2 752.462} C_VEL
LIN {X 0,Y 603.237,Z 602.81,A -85,B 0,C 180,E1 759.9,E2 759.9} C_VEL
LIN {X 0,Y 603.416,Z 602.81,A -85,B 0,C 180,E1 768.197,E2 768.197} C_VEL
LIN {X 0,Y 603.194,Z 602.81,A -85,B 0,C 180,E1 777.432,E2 777.432} C_VEL
LIN {X 0,Y 603.149,Z 602.81,A -85,B 0,C 180,E1 785.462,E2 785.462} C_VEL
LIN {X 0,Y 603.257,Z 602.81,A -85,B 0,C 180,E1 794.674,E2 794.674} C_VEL
LIN {X 0,Y 602.911,Z 602.81,A -85,B 0,C 180,E1 803.805,E2 803.805} C_VEL
LIN {X 0,Y 602.929,Z 602.81,A -85,B 0,C 180,E1 810.709,E2 810.709} C_VEL
LIN {X 0,Y 602.844,Z 602.81,A -85,B 0,C 180,E1 817.945,E2 817.945} C_VEL
LIN {X 0,Y 602.719,Z 602.81,A -85,B 0,C 180,E1 825.316,E2 825.316} C_VEL
LIN {X 0,Y 603.159,Z 602.81,A -85,B 0,C 180,E1 831.381,E2 831.381} C_VEL
LIN {X 0,Y 602.786,Z 602.81,A -85,B 0,C 180,E1 839.716,E2 839.716} C_VEL
LIN {X 0,Y 603.101,Z 602.81,A -85,B 0,C 180,E1 847.575,E2 847.575} C_VEL
LIN {X 0,Y 602.761,Z 602.81,A -85,B 0,C 180,E1 856.187,E2 856.187} C_VEL
LIN {X 0,Y 603.183,Z 602.81,A -85,B 0,C 180,E1 863.759,E2 863.759} C_VEL
LIN {X 0,Y 603.263,Z 602.81,A -85,B 0,C 180,E1 872.268,E2 872.268} C_VEL
LIN {X 0,Y 602.796,Z 603.976,A -85,B 0,C 180,E1 879.437,E2 879.437} C_VEL
LIN {X 0,Y 604.183,Z 659.574,A -85,B 0,C 180,E1 880.992,E2 880.992} C_VEL
LIN {X 0,Y 603.999,Z 708.685,A -85,B 0,C 180,E1 883.864,E2 883.864} C_VEL
LIN {X 0,Y 603.763,Z 748.28,A -85,B 0,C 180,E1 887.85,E2 887.85} C_VEL
LIN {X 0,Y 603.624,Z 775.655,A -85,B 0,C 180,E1 892.646,E2 892.646} C_VEL
LIN {X 0,Y 603.664,Z 788.789,A -85,B 0,C 180,E1 897.84,E2 897.84} C_VEL
LIN {X 0,Y 602.858,Z 789.832,A -85,B 0,C 180,E1 900.462,E2 900.462} C_VEL
LIN {X 0,Y 595.732,Z 786.244,A -85,B 0,C 180,E1 903.772,E2 903.772} C_VEL
LIN {X 0,Y 595.813,Z 769.307,A -85,B 0,C 180,E1 908.791,E2 908.791} C_VEL
LIN {X 0,Y 595.966,Z 738.406,A -85,B 0,C 180,E1 913.436,E2 913.436} C_VEL
LIN {X 0,Y 596.296,Z 696.496,A -85,B 0,C 180,E1 917.151,E2 917.151} C_VEL
LIN {X 0,Y 596.693,Z 645.138,A -85,B 0,C 180,E1 919.719,E2 919.719} C_VEL
LIN {X 0,Y 595.434,Z 602.81,A -85,B 0,C 180,E1 920.799,E2 920.799} C_VEL
LIN {X 0,Y 594.702,Z 602.81,A -85,B 0,C 180,E1 929.841,E2 929.841} C_VEL
LIN {X 0,Y 595.398,Z 602.81,A -85,B 0,C 180,E1 936.795,E2 936.795} C_VEL
LIN {X 0,Y 594.962,Z 602.81,A -85,B 0,C 180,E1 945.482,E2 945.482} C_VEL
LIN {X 0,Y 595.183,Z 602.81,A -85,B 0,C 180,E1 953.431,E2 953.431} C_VEL
LIN {X 0,Y 595.28,Z 602.81,A -85,B 0,C 180,E1 961.878,E2 961.878} C_VEL
LIN {X 0,Y 595.706,Z 604.465,A -85,B 0,C 180,E1 968.472,E2 968.472} C_VEL
LIN {X 0,Y 596.589,Z 697.307,A -85,B 0,C 180,E1 969.98,E2 969.98} C_VEL
LIN {X 0,Y 596.318,Z 749.021,A -85,B 0,C 180,E1 972.319,E2 972.319} C_VEL
LIN {X 0,Y 595.97,Z 792.14,A -85,B 0,C 180,E1 975.83,E2 975.83} C_VEL
LIN {X 0,Y 595.719,Z 823.822,A -85,B 0,C 180,E1 980.112,E2 980.112} C_VEL
LIN {X 0,Y 595.615,Z 843.256,A -85,B 0,C 180,E1 984.896,E2 984.896} C_VEL
LIN {X 0,Y 595.645,Z 849.842,A -85,B 0,C 180,E1 989.282,E2 989.282} C_VEL
LIN {X 0,Y 595.738,Z 845.026,A -85,B 0,C 180,E1 994.394,E2 994.394} C_VEL
LIN {X 0,Y 595.901,Z 825.672,A -85,B 0,C 180,E1 999.539,E2 999.539} C_VEL
LIN {X 0,Y 596.014,Z 793.637,A -85,B 0,C 180,E1 1004.008,E2 1004.008} C_VEL
LIN {X 0,Y 596.355,Z 749.532,A -85,B 0,C 180,E1 1007.648,E2 1007.648} C_VEL
LIN {X 0,Y 596.661,Z 697.952,A -85,B 0,C 180,E1 1009.998,E2 1009.998} C_VEL
LIN {X 0,Y 595.515,Z 602.81,A -85,B 0,C 180,E1 1011.695,E2 1011.695} C_VEL
LIN {X 0,Y 594.763,Z 602.81,A -85,B 0,C 180,E1 1019.847,E2 1019.847} C_VEL
LIN {X 0,Y 595.456,Z 602.81,A -85,B 0,C 180,E1 1026.801,E2 1026.801} C_VEL
LIN {X 0,Y 595.034,Z 602.81,A -85,B 0,C 180,E1 1035.466,E2 1035.466} C_VEL
LIN {X 0,Y 595.243,Z 602.81,A -85,B 0,C 180,E1 1043.436,E2 1043.436} C_VEL
LIN {X 0,Y 595.189,Z 602.81,A -85,B 0,C 180,E1 1051.856,E2 1051.856} C_VEL
LIN {X 0,Y 594.842,Z 602.81,A -85,B 0,C 180,E1 1061.403,E2 1061.403} C_VEL
LIN {X 0,Y 595.917,Z 604.419,A -85,B 0,C 180,E1 1067.775,E2 1067.775} C_VEL
LIN {X 0,Y 595.887,Z 644.56,A -85,B 0,C 180,E1 1069.638,E2 1069.638} C_VEL
LIN {X 0,Y 595.359,Z 675.97,A -85,B 0,C 180,E1 1072.677,E2 1072.677} C_VEL
LIN {X 0,Y 595.2,Z 694.464,A -85,B 0,C 180,E1 1076.344,E2 1076.344} C_VEL
LIN {X 0,Y 595.825,Z 699.789,A -85,B 0,C 180,E1 1079.269,E2 1079.269} C_VEL
LIN {X 0,Y 595.691,Z 694.191,A -85,B 0,C 180,E1 1083.65,E2 1083.65} C_VEL
LIN {X 0,Y 595.814,Z 673.896,A -85,B 0,C 180,E1 1087.504,E2 1087.504} C_VEL
LIN {X 0,Y 596.029,Z 641.861,A -85,B 0,C 180,E1 1090.45,E2 1090.45} C_VEL
LIN {X 0,Y 595.772,Z 602.81,A -85,B 0,C 180,E1 1092.333,E2 1092.333} C_VEL
LIN {X 0,Y 595.152,Z 602.81,A -85,B 0,C 180,E1 1101.697,E2 1101.697} C_VEL
LIN {X 0,Y 595.11,Z 602.81,A -85,B 0,C 180,E1 1111.514,E2 1111.514} C_VEL
LIN {X 0,Y 594.655,Z 602.81,A -85,B 0,C 180,E1 1121.154,E2 1121.154} C_VEL
LIN {X 0,Y 594.684,Z 602.81,A -85,B 0,C 180,E1 1129.394,E2 1129.394} C_VEL
LIN {X 0,Y 594.7,Z 602.81,A -85,B 0,C 180,E1 1138.449,E2 1138.449} C_VEL
LIN {X 0,Y 594.471,Z 602.81,A -85,B 0,C 180,E1 1146.682,E2 1146.682} C_VEL
LIN {X 0,Y 595.263,Z 602.81,A -85,B 0,C 180,E1 1154.463,E2 1154.463} C_VEL
LIN {X 0,Y 595.048,Z 602.81,A -85,B 0,C 180,E1 1163.399,E2 1163.399} C_VEL
LIN {X 0,Y 594.938,Z 602.81,A -85,B 0,C 180,E1 1170.719,E2 1170.719} C_VEL
LIN {X 0,Y 594.814,Z 602.81,A -85,B 0,C 180,E1 1178.053,E2 1178.053} C_VEL
LIN {X 0,Y 594.675,Z 602.81,A -85,B 0,C 180,E1 1185.528,E2 1185.528} C_VEL
LIN {X 0,Y 595.005,Z 602.81,A -85,B 0,C 180,E1 1191.689,E2 1191.689} C_VEL
LIN {X 0,Y 594.754,Z 602.81,A -85,B 0,C 180,E1 1199.82,E2 1199.82} C_VEL
LIN {X 0,Y 595.443,Z 602.81,A -85,B 0,C 180,E1 1206.772,E2 1206.772} C_VEL
LIN {X 0,Y 595.023,Z 602.81,A -85,B 0,C 180,E1 1215.468,E2 1215.468} C_VEL
LIN {X 0,Y 595.258,Z 602.81,A -85,B 0,C 180,E1 1223.394,E2 1223.394} C_VEL
LIN {X 0,Y 595.21,Z 602.81,A -85,B 0,C 180,E1 1231.86,E2 1231.86} C_VEL
LIN {X 0,Y 595.205,Z 604.254,A -85,B 0,C 180,E1 1239.167,E2 1239.167} C_VEL
LIN {X 0,Y 596.548,Z 658.839,A -85,B 0,C 180,E1 1240.708,E2 1240.708} C_VEL
LIN {X 0,Y 596.247,Z 707.437,A -85,B 0,C 180,E1 1243.554,E2 1243.554} C_VEL
LIN {X 0,Y 595.801,Z 748.032,A -85,B 0,C 180,E1 1247.653,E2 1247.653} C_VEL
LIN {X 0,Y 595.528,Z 775.084,A -85,B 0,C 180,E1 1252.408,E2 1252.408} C_VEL
LIN {X 0,Y 595.637,Z 788.792,A -85,B 0,C 180,E1 1257.811,E2 1257.811} C_VEL
LIN {X 0,Y 595.517,Z 787.727,A -85,B 0,C 180,E1 1262.922,E2 1262.922} C_VEL
LIN {X 0,Y 595.732,Z 786.244,A -85,B 0,C 180,E1 1263.772,E2 1263.772} C_VEL
LIN {X 0,Y 587.166,Z 777.438,A -85,B 0,C 180,E1 1266.993,E2 1266.993} C_VEL
LIN {X 0,Y 587.488,Z 752.979,A -85,B 0,C 180,E1 1271.738,E2 1271.738} C_VEL
LIN {X 0,Y 588.142,Z 714.495,A -85,B 0,C 180,E1 1276.008,E2 1276.008} C_VEL
LIN {X 0,Y 588.893,Z 667.05,A -85,B 0,C 180,E1 1279.088,E2 1279.088} C_VEL
LIN {X 0,Y 589.293,Z 612.808,A -85,B 0,C 180,E1 1280.828,E2 1280.828} C_VEL
LIN {X 0,Y 587.285,Z 602.81,A -85,B 0,C 180,E1 1281.065,E2 1281.065} C_VEL
LIN {X 0,Y 586.555,Z 602.81,A -85,B 0,C 180,E1 1290.298,E2 1290.298} C_VEL
LIN {X 0,Y 586.831,Z 602.81,A -85,B 0,C 180,E1 1297.962,E2 1297.962} C_VEL
LIN {X 0,Y 587.024,Z 602.81,A -85,B 0,C 180,E1 1305.309,E2 1305.309} C_VEL
LIN {X 0,Y 586.69,Z 602.81,A -85,B 0,C 180,E1 1314.565,E2 1314.565} C_VEL
LIN {X 0,Y 586.931,Z 602.81,A -85,B 0,C 180,E1 1323.125,E2 1323.125} C_VEL
LIN {X 0,Y 587.615,Z 604.671,A -85,B 0,C 180,E1 1328.163,E2 1328.163} C_VEL
LIN {X 0,Y 589.074,Z 696.973,A -85,B 0,C 180,E1 1329.704,E2 1329.704} C_VEL
LIN {X 0,Y 588.592,Z 749.323,A -85,B 0,C 180,E1 1332.098,E2 1332.098} C_VEL
LIN {X 0,Y 588.13,Z 792.364,A -85,B 0,C 180,E1 1335.662,E2 1335.662} C_VEL
LIN {X 0,Y 587.637,Z 825.802,A -85,B 0,C 180,E1 1340.35,E2 1340.35} C_VEL
LIN {X 0,Y 587.303,Z 845.077,A -85,B 0,C 180,E1 1345.567,E2 1345.567} C_VEL
LIN {X 0,Y 587.237,Z 849.836,A -85,B 0,C 180,E1 1350.752,E2 1350.752} C_VEL
LIN {X 0,Y 587.243,Z 841.538,A -85,B 0,C 180,E1 1355.797,E2 1355.797} C_VEL
LIN {X 0,Y 587.507,Z 819.441,A -85,B 0,C 180,E1 1360.783,E2 1360.783} C_VEL
LIN {X 0,Y 588.039,Z 783.796,A -85,B 0,C 180,E1 1365.215,E2 1365.215} C_VEL
LIN {X 0,Y 588.78,Z 737.295,A -85,B 0,C 180,E1 1368.61,E2 1368.61} C_VEL
LIN {X 0,Y 589.305,Z 685.112,A -85,B 0,C 180,E1 1370.612,E2 1370.612} C_VEL
LIN {X 0,Y 587.376,Z 602.81,A -85,B 0,C 180,E1 1372.011,E2 1372.011} C_VEL
LIN {X 0,Y 586.607,Z 602.81,A -85,B 0,C 180,E1 1380.306,E2 1380.306} C_VEL
LIN {X 0,Y 586.875,Z 602.81,A -85,B 0,C 180,E1 1387.94,E2 1387.94} C_VEL
LIN {X 0,Y 586.567,Z 602.81,A -85,B 0,C 180,E1 1396.718,E2 1396.718} C_VEL
LIN {X 0,Y 586.731,Z 602.81,A -85,B 0,C 180,E1 1404.571,E2 1404.571} C_VEL
LIN {X 0,Y 586.736,Z 602.81,A -85,B 0,C 180,E1 1413.178,E2 1413.178} C_VEL
LIN {X 0,Y 586.906,Z 602.81,A -85,B 0,C 180,E1 1421.143,E2 1421.143} C_VEL
LIN {X 0,Y 587.696,Z 603.927,A -85,B 0,C 180,E1 1427.589,E2 1427.589} C_VEL
LIN {X 0,Y 588.011,Z 644.547,A -85,B 0,C 180,E1 1429.497,E2 1429.497} C_VEL
LIN {X 0,Y 587.438,Z 675.967,A -85,B 0,C 180,E1 1432.578,E2 1432.578} C_VEL
LIN {X 0,Y 587.217,Z 694.458,A -85,B 0,C 180,E1 1436.295,E2 1436.295} C_VEL
LIN {X 0,Y 587.811,Z 699.786,A -85,B 0,C 180,E1 1439.259,E2 1439.259} C_VEL
LIN {X 0,Y 587.665,Z 694.187,A -85,B 0,C 180,E1 1443.7,E2 1443.7} C_VEL
LIN {X 0,Y 587.818,Z 673.926,A -85,B 0,C 180,E1 1447.602,E2 1447.602} C_VEL
LIN {X 0,Y 588.137,Z 641.854,A -85,B 0,C 180,E1 1450.592,E2 1450.592} C_VEL
LIN {X 0,Y 587.745,Z 602.81,A -85,B 0,C 180,E1 1452.487,E2 1452.487} C_VEL
LIN {X 0,Y 587.178,Z 602.81,A -85,B 0,C 180,E1 1462.006,E2 1462.006} C_VEL
LIN {X 0,Y 586.816,Z 602.81,A -85,B 0,C 180,E1 1472.012,E2 1472.012} C_VEL
LIN {X 0,Y 586.614,Z 602.81,A -85,B 0,C 180,E1 1481.271,E2 1481.271} C_VEL
LIN {X 0,Y 587.061,Z 602.81,A -85,B 0,C 180,E1 1488.753,E2 1488.753} C_VEL
LIN {X 0,Y 586.77,Z 602.81,A -85,B 0,C 180,E1 1497.972,E2 1497.972} C_VEL
LIN {X 0,Y 586.452,Z 602.81,A -85,B 0,C 180,E1 1506.717,E2 1506.717} C_VEL
LIN {X 0,Y 587.241,Z 602.81,A -85,B 0,C 180,E1 1514.245,E2 1514.245} C_VEL
LIN {X 0,Y 587.072,Z 602.81,A -85,B 0,C 180,E1 1523.309,E2 1523.309} C_VEL
LIN {X 0,Y 586.933,Z 602.81,A -85,B 0,C 180,E1 1530.729,E2 1530.729} C_VEL
LIN {X 0,Y 586.8,Z 602.81,A -85,B 0,C 180,E1 1538.164,E2 1538.164} C_VEL
LIN {X 0,Y 586.641,Z 602.81,A -85,B 0,C 180,E1 1545.746,E2 1545.746} C_VEL
LIN {X 0,Y 586.563,Z 602.81,A -85,B 0,C 180,E1 1553.309,E2 1553.309} C_VEL
LIN {X 0,Y 586.604,Z 602.81,A -85,B 0,C 180,E1 1560.278,E2 1560.278} C_VEL
LIN {X 0,Y 586.881,Z 602.81,A -85,B 0,C 180,E1 1567.945,E2 1567.945} C_VEL
LIN {X 0,Y 587.085,Z 602.81,A -85,B 0,C 180,E1 1575.279,E2 1575.279} C_VEL
LIN {X 0,Y 586.716,Z 602.81,A -85,B 0,C 180,E1 1584.532,E2 1584.532} C_VEL
LIN {X 0,Y 586.783,Z 602.81,A -85,B 0,C 180,E1 1593.116,E2 1593.116} C_VEL
LIN {X 0,Y 587.238,Z 602.81,A -85,B 0,C 180,E1 1598.852,E2 1598.852} C_VEL
LIN {X 0,Y 588.943,Z 657.474,A -85,B 0,C 180,E1 1600.393,E2 1600.393} C_VEL
LIN {X 0,Y 588.474,Z 706.18,A -85,B 0,C 180,E1 1603.234,E2 1603.234} C_VEL
LIN {X 0,Y 587.794,Z 746.824,A -85,B 0,C 180,E1 1607.325,E2 1607.325} C_VEL
LIN {X 0,Y 587.463,Z 774.688,A -85,B 0,C 180,E1 1612.207,E2 1612.207} C_VEL
LIN {X 0,Y 587.385,Z 788.194,A -85,B 0,C 180,E1 1617.294,E2 1617.294} C_VEL
LIN {X 0,Y 587.532,Z 787.731,A -85,B 0,C 180,E1 1622.962,E2 1622.962} C_VEL
LIN {X 0,Y 587.166,Z 777.438,A -85,B 0,C 180,E1 1626.993,E2 1626.993} C_VEL
LIN {X 0,Y 579.468,Z 763.71,A -85,B 0,C 180,E1 1630.14,E2 1630.14} C_VEL
LIN {X 0,Y 580.053,Z 730.432,A -85,B 0,C 180,E1 1634.709,E2 1634.709} C_VEL
LIN {X 0,Y 580.947,Z 685.173,A -85,B 0,C 180,E1 1638.366,E2 1638.366} C_VEL
LIN {X 0,Y 581.714,Z 633.711,A -85,B 0,C 180,E1 1640.621,E2 1640.621} C_VEL
LIN {X 0,Y 579.119,Z 602.81,A -85,B 0,C 180,E1 1641.396,E2 1641.396} C_VEL
LIN {X 0,Y 579.004,Z 602.81,A -85,B 0,C 180,E1 1649.004,E2 1649.004} C_VEL
LIN {X 0,Y 578.814,Z 602.81,A -85,B 0,C 180,E1 1658.033,E2 1658.033} C_VEL
LIN {X 0,Y 578.683,Z 602.81,A -85,B 0,C 180,E1 1666.15,E2 1666.15} C_VEL
LIN {X 0,Y 578.768,Z 602.81,A -85,B 0,C 180,E1 1673.866,E2 1673.866} C_VEL
LIN {X 0,Y 578.967,Z 602.81,A -85,B 0,C 180,E1 1682.714,E2 1682.714} C_VEL
LIN {X 0,Y 579.378,Z 604.282,A -85,B 0,C 180,E1 1687.832,E2 1687.832} C_VEL
LIN {X 0,Y 581.539,Z 697.457,A -85,B 0,C 180,E1 1689.444,E2 1689.444} C_VEL
LIN {X 0,Y 580.91,Z 749.19,A -85,B 0,C 180,E1 1691.844,E2 1691.844} C_VEL
LIN {X 0,Y 580.279,Z 792.741,A -85,B 0,C 180,E1 1695.505,E2 1695.505} C_VEL
LIN {X 0,Y 579.698,Z 825.803,A -85,B 0,C 180,E1 1700.217,E2 1700.217} C_VEL
LIN {X 0,Y 579.35,Z 845.076,A -85,B 0,C 180,E1 1705.506,E2 1705.506} C_VEL
LIN {X 0,Y 579.243,Z 849.836,A -85,B 0,C 180,E1 1710.763,E2 1710.763} C_VEL
LIN {X 0,Y 579.201,Z 841.539,A -85,B 0,C 180,E1 1715.877,E2 1715.877} C_VEL
LIN {X 0,Y 579.487,Z 818.752,A -85,B 0,C 180,E1 1721.048,E2 1721.048} C_VEL
LIN {X 0,Y 580.158,Z 782.686,A -85,B 0,C 180,E1 1725.534,E2 1725.534} C_VEL
LIN {X 0,Y 581.14,Z 735.478,A -85,B 0,C 180,E1 1728.963,E2 1728.963} C_VEL
LIN {X 0,Y 581.827,Z 682.911,A -85,B 0,C 180,E1 1730.944,E2 1730.944} C_VEL
LIN {X 0,Y 579.306,Z 602.81,A -85,B 0,C 180,E1 1732.239,E2 1732.239} C_VEL
LIN {X 0,Y 578.473,Z 602.81,A -85,B 0,C 180,E1 1740.778,E2 1740.778} C_VEL
LIN {X 0,Y 578.854,Z 602.81,A -85,B 0,C 180,E1 1748.041,E2 1748.041} C_VEL
LIN {X 0,Y 578.751,Z 602.81,A -85,B 0,C 180,E1 1756.154,E2 1756.154} C_VEL
LIN {X 0,Y 578.823,Z 602.81,A -85,B 0,C 180,E1 1763.851,E2 1763.851} C_VEL
LIN {X 0,Y 578.8,Z 602.81,A -85,B 0,C 180,E1 1772.688,E2 1772.688} C_VEL
LIN {X 0,Y 579.019,Z 602.81,A -85,B 0,C 180,E1 1780.876,E2 1780.876} C_VEL
LIN {X 0,Y 579.696,Z 604.466,A -85,B 0,C 180,E1 1787.431,E2 1787.431} C_VEL
LIN {X 0,Y 580.13,Z 644.146,A -85,B 0,C 180,E1 1789.326,E2 1789.326} C_VEL
LIN {X 0,Y 579.506,Z 675.964,A -85,B 0,C 180,E1 1792.476,E2 1792.476} C_VEL
LIN {X 0,Y 579.249,Z 694.452,A -85,B 0,C 180,E1 1796.244,E2 1796.244} C_VEL
LIN {X 0,Y 579.813,Z 699.778,A -85,B 0,C 180,E1 1799.249,E2 1799.249} C_VEL
LIN {X 0,Y 579.642,Z 694.181,A -85,B 0,C 180,E1 1803.751,E2 1803.751} C_VEL
LIN {X 0,Y 579.826,Z 673.919,A -85,B 0,C 180,E1 1807.707,E2 1807.707} C_VEL
LIN {X 0,Y 580.24,Z 641.633,A -85,B 0,C 180,E1 1810.752,E2 1810.752} C_VEL
LIN {X 0,Y 579.732,Z 602.81,A -85,B 0,C 180,E1 1812.662,E2 1812.662} C_VEL
LIN {X 0,Y 579.181,Z 602.81,A -85,B 0,C 180,E1 1822.327,E2 1822.327} C_VEL
LIN {X 0,Y 578.866,Z 602.81,A -85,B 0,C 180,E1 1831.557,E2 1831.557} C_VEL
LIN {X 0,Y 578.905,Z 602.81,A -85,B 0,C 180,E1 1839.956,E2 1839.956} C_VEL
LIN {X 0,Y 579.167,Z 602.81,A -85,B 0,C 180,E1 1848.306,E2 1848.306} C_VEL
LIN {X 0,Y 578.594,Z 602.81,A -85,B 0,C 180,E1 1858.469,E2 1858.469} C_VEL
LIN {X 0,Y 578.669,Z 602.81,A -85,B 0,C 180,E1 1866.006,E2 1866.006} C_VEL
LIN {X 0,Y 579.2,Z 602.81,A -85,B 0,C 180,E1 1874.021,E2 1874.021} C_VEL
LIN {X 0,Y 579.093,Z 602.81,A -85,B 0,C 180,E1 1883.216,E2 1883.216} C_VEL
LIN {X 0,Y 578.953,Z 602.81,A -85,B 0,C 180,E1 1890.739,E2 1890.739} C_VEL
LIN {X 0,Y 578.774,Z 602.81,A -85,B 0,C 180,E1 1898.278,E2 1898.278} C_VEL
LIN {X 0,Y 578.614,Z 602.81,A -85,B 0,C 180,E1 1905.97,E2 1905.97} C_VEL
LIN {X 0,Y 578.779,Z 602.81,A -85,B 0,C 180,E1 1912.329,E2 1912.329} C_VEL
LIN {X 0,Y 578.466,Z 602.81,A -85,B 0,C 180,E1 1920.749,E2 1920.749} C_VEL
LIN {X 0,Y 578.865,Z 602.81,A -85,B 0,C 180,E1 1928.009,E2 1928.009} C_VEL
LIN {X 0,Y 578.743,Z 602.81,A -85,B 0,C 180,E1 1936.119,E2 1936.119} C_VEL
LIN {X 0,Y 578.797,Z 602.81,A -85,B 0,C 180,E1 1943.852,E2 1943.852} C_VEL
LIN {X 0,Y 578.841,Z 602.81,A -85,B 0,C 180,E1 1952.693,E2 1952.693} C_VEL
LIN {X 0,Y 579.428,Z 604.172,A -85,B 0,C 180,E1 1958.573,E2 1958.573} C_VEL
LIN {X 0,Y 581.383,Z 656.944,A -85,B 0,C 180,E1 1960.106,E2 1960.106} C_VEL
LIN {X 0,Y 580.701,Z 706.178,A -85,B 0,C 180,E1 1963.003,E2 1963.003} C_VEL
LIN {X 0,Y 579.862,Z 746.823,A -85,B 0,C 180,E1 1967.149,E2 1967.149} C_VEL
LIN {X 0,Y 579.45,Z 774.689,A -85,B 0,C 180,E1 1972.099,E2 1972.099} C_VEL
LIN {X 0,Y 579.408,Z 788.275,A -85,B 0,C 180,E1 1977.324,E2 1977.324} C_VEL
LIN {X 0,Y 579.555,Z 787.735,A -85,B 0,C 180,E1 1983.003,E2 1983.003} C_VEL
LIN {X 0,Y 579.772,Z 772.745,A -85,B 0,C 180,E1 1988.278,E2 1988.278} C_VEL
LIN {X 0,Y 579.468,Z 763.71,A -85,B 0,C 180,E1 1990.14,E2 1990.14} C_VEL
LIN {X 0,Y 572.187,Z 745.661,A -85,B 0,C 180,E1 1993.09,E2 1993.09} C_VEL
LIN {X 0,Y 572.93,Z 705.691,A -85,B 0,C 180,E1 1997.184,E2 1997.184} C_VEL
LIN {X 0,Y 573.874,Z 655.828,A -85,B 0,C 180,E1 2000.122,E2 2000.122} C_VEL
LIN {X 0,Y 572.395,Z 607.882,A -85,B 0,C 180,E1 2001.557,E2 2001.557} C_VEL
LIN {X 0,Y 570.897,Z 602.81,A -85,B 0,C 180,E1 2001.879,E2 2001.879} C_VEL
LIN {X 0,Y 570.558,Z 602.81,A -85,B 0,C 180,E1 2010.22,E2 2010.22} C_VEL
LIN {X 0,Y 570.626,Z 602.81,A -85,B 0,C 180,E1 2018.679,E2 2018.679} C_VEL
LIN {X 0,Y 570.348,Z 602.81,A -85,B 0,C 180,E1 2027.298,E2 2027.298} C_VEL
LIN {X 0,Y 570.395,Z 602.81,A -85,B 0,C 180,E1 2035.13,E2 2035.13} C_VEL
LIN {X 0,Y 570.725,Z 602.81,A -85,B 0,C 180,E1 2043.994,E2 2043.994} C_VEL
LIN {X 0,Y 571.356,Z 604.586,A -85,B 0,C 180,E1 2047.507,E2 2047.507} C_VEL
LIN {X 0,Y 574.371,Z 645.245,A -85,B 0,C 180,E1 2048.169,E2 2048.169} C_VEL
LIN {X 0,Y 574,Z 706.284,A -85,B 0,C 180,E1 2049.463,E2 2049.463} C_VEL
LIN {X 0,Y 572.972,Z 757.894,A -85,B 0,C 180,E1 2052.183,E2 2052.183} C_VEL
LIN {X 0,Y 572.005,Z 800.514,A -85,B 0,C 180,E1 2056.2,E2 2056.2} C_VEL
LIN {X 0,Y 571.452,Z 829.581,A -85,B 0,C 180,E1 2060.845,E2 2060.845} C_VEL
LIN {X 0,Y 571.371,Z 845.076,A -85,B 0,C 180,E1 2065.443,E2 2065.443} C_VEL
LIN {X 0,Y 571.239,Z 849.835,A -85,B 0,C 180,E1 2070.773,E2 2070.773} C_VEL
LIN {X 0,Y 571.131,Z 841.084,A -85,B 0,C 180,E1 2076.113,E2 2076.113} C_VEL
LIN {X 0,Y 571.54,Z 818.29,A -85,B 0,C 180,E1 2081.278,E2 2081.278} C_VEL
LIN {X 0,Y 572.353,Z 781.642,A -85,B 0,C 180,E1 2085.85,E2 2085.85} C_VEL
LIN {X 0,Y 573.493,Z 735.481,A -85,B 0,C 180,E1 2089.226,E2 2089.226} C_VEL
LIN {X 0,Y 574.369,Z 681.702,A -85,B 0,C 180,E1 2091.259,E2 2091.259} C_VEL
LIN {X 0,Y 571.764,Z 605.681,A -85,B 0,C 180,E1 2092.461,E2 2092.461} C_VEL
LIN {X 0,Y 571.16,Z 602.81,A -85,B 0,C 180,E1 2092.67,E2 2092.67} C_VEL
LIN {X 0,Y 570.429,Z 602.81,A -85,B 0,C 180,E1 2101.26,E2 2101.26} C_VEL
LIN {X 0,Y 570.644,Z 602.81,A -85,B 0,C 180,E1 2108.689,E2 2108.689} C_VEL
LIN {X 0,Y 570.401,Z 602.81,A -85,B 0,C 180,E1 2117.28,E2 2117.28} C_VEL
LIN {X 0,Y 570.443,Z 602.81,A -85,B 0,C 180,E1 2125.113,E2 2125.113} C_VEL
LIN {X 0,Y 570.475,Z 602.81,A -85,B 0,C 180,E1 2133.965,E2 2133.965} C_VEL
LIN {X 0,Y 570.563,Z 602.81,A -85,B 0,C 180,E1 2142.189,E2 2142.189} C_VEL
LIN {X 0,Y 571.55,Z 604.401,A -85,B 0,C 180,E1 2147.249,E2 2147.249} C_VEL
LIN {X 0,Y 572.271,Z 644.024,A -85,B 0,C 180,E1 2149.17,E2 2149.17} C_VEL
LIN {X 0,Y 571.556,Z 675.959,A -85,B 0,C 180,E1 2152.37,E2 2152.37} C_VEL
LIN {X 0,Y 571.267,Z 694.442,A -85,B 0,C 180,E1 2156.191,E2 2156.191} C_VEL
LIN {X 0,Y 571.799,Z 699.769,A -85,B 0,C 180,E1 2159.239,E2 2159.239} C_VEL
LIN {X 0,Y 571.62,Z 694.175,A -85,B 0,C 180,E1 2163.804,E2 2163.804} C_VEL
LIN {X 0,Y 571.859,Z 673.911,A -85,B 0,C 180,E1 2167.815,E2 2167.815} C_VEL
LIN {X 0,Y 572.362,Z 641.234,A -85,B 0,C 180,E1 2170.929,E2 2170.929} C_VEL
LIN {X 0,Y 571.672,Z 602.81,A -85,B 0,C 180,E1 2172.844,E2 2172.844} C_VEL
LIN {X 0,Y 571.071,Z 602.81,A -85,B 0,C 180,E1 2183.524,E2 2183.524} C_VEL
LIN {X 0,Y 570.921,Z 602.81,A -85,B 0,C 180,E1 2191.217,E2 2191.217} C_VEL
LIN {X 0,Y 570.668,Z 602.81,A -85,B 0,C 180,E1 2200.711,E2 2200.711} C_VEL
LIN {X 0,Y 570.65,Z 602.81,A -85,B 0,C 180,E1 2209.332,E2 2209.332} C_VEL
LIN {X 0,Y 570.541,Z 602.81,A -85,B 0,C 180,E1 2218.747,E2 2218.747} C_VEL
LIN {X 0,Y 570.423,Z 602.81,A -85,B 0,C 180,E1 2226.602,E2 2226.602} C_VEL
LIN {X 0,Y 570.825,Z 602.81,A -85,B 0,C 180,E1 2235.36,E2 2235.36} C_VEL
LIN {X 0,Y 571.14,Z 602.81,A -85,B 0,C 180,E1 2243.121,E2 2243.121} C_VEL
LIN {X 0,Y 570.947,Z 602.81,A -85,B 0,C 180,E1 2250.749,E2 2250.749} C_VEL
LIN {X 0,Y 570.754,Z 602.81,A -85,B 0,C 180,E1 2258.395,E2 2258.395} C_VEL
LIN {X 0,Y 570.595,Z 602.81,A -85,B 0,C 180,E1 2266.201,E2 2266.201} C_VEL
LIN {X 0,Y 570.516,Z 602.81,A -85,B 0,C 180,E1 2274.332,E2 2274.332} C_VEL
LIN {X 0,Y 570.404,Z 602.81,A -85,B 0,C 180,E1 2281.232,E2 2281.232} C_VEL
LIN {X 0,Y 570.67,Z 602.81,A -85,B 0,C 180,E1 2288.655,E2 2288.655} C_VEL
LIN {X 0,Y 570.395,Z 602.81,A -85,B 0,C 180,E1 2297.283,E2 2297.283} C_VEL
LIN {X 0,Y 570.413,Z 602.81,A -85,B 0,C 180,E1 2305.114,E2 2305.114} C_VEL
LIN {X 0,Y 570.531,Z 602.81,A -85,B 0,C 180,E1 2313.97,E2 2313.97} C_VEL
LIN {X 0,Y 571.265,Z 604.156,A -85,B 0,C 180,E1 2318.251,E2 2318.251} C_VEL
LIN {X 0,Y 573.898,Z 652.551,A -85,B 0,C 180,E1 2319.653,E2 2319.653} C_VEL
LIN {X 0,Y 573.002,Z 702.901,A -85,B 0,C 180,E1 2322.508,E2 2322.508} C_VEL
LIN {X 0,Y 571.883,Z 743.881,A -85,B 0,C 180,E1 2326.578,E2 2326.578} C_VEL
LIN {X 0,Y 571.269,Z 771.495,A -85,B 0,C 180,E1 2331.216,E2 2331.216} C_VEL
LIN {X 0,Y 571.061,Z 786.661,A -85,B 0,C 180,E1 2336.192,E2 2336.192} C_VEL
LIN {X 0,Y 570.833,Z 789.818,A -85,B 0,C 180,E1 2340.763,E2 2340.763} C_VEL
LIN {X 0,Y 571.033,Z 782.123,A -85,B 0,C 180,E1 2345.72,E2 2345.72} C_VEL
LIN {X 0,Y 571.422,Z 761.586,A -85,B 0,C 180,E1 2350.667,E2 2350.667} C_VEL
LIN {X 0,Y 572.187,Z 745.661,A -85,B 0,C 180,E1 2353.09,E2 2353.09} C_VEL
LIN {X 0,Y 564.462,Z 723.912,A -85,B 0,C 180,E1 2355.811,E2 2355.811} C_VEL
LIN {X 0,Y 565.894,Z 676.675,A -85,B 0,C 180,E1 2359.382,E2 2359.382} C_VEL
LIN {X 0,Y 566.862,Z 623.509,A -85,B 0,C 180,E1 2361.464,E2 2361.464} C_VEL
LIN {X 0,Y 562.806,Z 602.81,A -85,B 0,C 180,E1 2362.118,E2 2362.118} C_VEL
LIN {X 0,Y 562.653,Z 602.81,A -85,B 0,C 180,E1 2369.932,E2 2369.932} C_VEL
LIN {X 0,Y 562.846,Z 602.81,A -85,B 0,C 180,E1 2377.347,E2 2377.347} C_VEL
LIN {X 0,Y 562.476,Z 602.81,A -85,B 0,C 180,E1 2386.553,E2 2386.553} C_VEL
LIN {X 0,Y 562.323,Z 602.81,A -85,B 0,C 180,E1 2395.395,E2 2395.395} C_VEL
LIN {X 0,Y 562.77,Z 602.81,A -85,B 0,C 180,E1 2403.599,E2 2403.599} C_VEL
LIN {X 0,Y 563.066,Z 603.505,A -85,B 0,C 180,E1 2407.143,E2 2407.143} C_VEL
LIN {X 0,Y 566.641,Z 627.758,A -85,B 0,C 180,E1 2407.621,E2 2407.621} C_VEL
LIN {X 0,Y 566.533,Z 700.305,A -85,B 0,C 180,E1 2408.963,E2 2408.963} C_VEL
LIN {X 0,Y 565.506,Z 752.242,A -85,B 0,C 180,E1 2411.535,E2 2411.535} C_VEL
LIN {X 0,Y 564.546,Z 794.97,A -85,B 0,C 180,E1 2415.345,E2 2415.345} C_VEL
LIN {X 0,Y 563.847,Z 825.806,A -85,B 0,C 180,E1 2419.939,E2 2419.939} C_VEL
LIN {X 0,Y 563.35,Z 845.271,A -85,B 0,C 180,E1 2425.475,E2 2425.475} C_VEL
LIN {X 0,Y 563.235,Z 849.835,A -85,B 0,C 180,E1 2430.784,E2 2430.784} C_VEL
LIN {X 0,Y 563.117,Z 841.085,A -85,B 0,C 180,E1 2436.2,E2 2436.2} C_VEL
LIN {X 0,Y 563.593,Z 818.798,A -85,B 0,C 180,E1 2441.356,E2 2441.356} C_VEL
LIN {X 0,Y 564.488,Z 784.372,A -85,B 0,C 180,E1 2445.806,E2 2445.806} C_VEL
LIN {X 0,Y 565.83,Z 738.994,A -85,B 0,C 180,E1 2449.293,E2 2449.293} C_VEL
LIN {X 0,Y 566.86,Z 686.824,A -85,B 0,C 180,E1 2451.423,E2 2451.423} C_VEL
LIN {X 0,Y 564.29,Z 606.911,A -85,B 0,C 180,E1 2452.758,E2 2452.758} C_VEL
LIN {X 0,Y 563.089,Z 602.81,A -85,B 0,C 180,E1 2453.014,E2 2453.014} C_VEL
LIN {X 0,Y 562.357,Z 602.81,A -85,B 0,C 180,E1 2461.786,E2 2461.786} C_VEL
LIN {X 0,Y 562.477,Z 602.81,A -85,B 0,C 180,E1 2469.744,E2 2469.744} C_VEL
LIN {X 0,Y 562.324,Z 602.81,A -85,B 0,C 180,E1 2477.925,E2 2477.925} C_VEL
LIN {X 0,Y 562.36,Z 602.81,A -85,B 0,C 180,E1 2485.403,E2 2485.403} C_VEL
LIN {X 0,Y 562.548,Z 602.81,A -85,B 0,C 180,E1 2493.57,E2 2493.57} C_VEL
LIN {X 0,Y 562.612,Z 602.81,A -85,B 0,C 180,E1 2501.929,E2 2501.929} C_VEL
LIN {X 0,Y 563.41,Z 604.334,A -85,B 0,C 180,E1 2507.061,E2 2507.061} C_VEL
LIN {X 0,Y 564.419,Z 643.061,A -85,B 0,C 180,E1 2508.953,E2 2508.953} C_VEL
LIN {X 0,Y 563.731,Z 674.538,A -85,B 0,C 180,E1 2512.069,E2 2512.069} C_VEL
LIN {X 0,Y 563.286,Z 694.432,A -85,B 0,C 180,E1 2516.137,E2 2516.137} C_VEL
LIN {X 0,Y 563.812,Z 699.759,A -85,B 0,C 180,E1 2519.228,E2 2519.228} C_VEL
LIN {X 0,Y 563.629,Z 694.169,A -85,B 0,C 180,E1 2523.858,E2 2523.858} C_VEL
LIN {X 0,Y 563.859,Z 673.904,A -85,B 0,C 180,E1 2527.927,E2 2527.927} C_VEL
LIN {X 0,Y 564.471,Z 641.353,A -85,B 0,C 180,E1 2531.075,E2 2531.075} C_VEL
LIN {X 0,Y 563.66,Z 602.81,A -85,B 0,C 180,E1 2533.029,E2 2533.029} C_VEL
LIN {X 0,Y 563.085,Z 602.81,A -85,B 0,C 180,E1 2543.001,E2 2543.001} C_VEL
LIN {X 0,Y 562.709,Z 602.81,A -85,B 0,C 180,E1 2551.829,E2 2551.829} C_VEL
LIN {X 0,Y 562.487,Z 602.81,A -85,B 0,C 180,E1 2561.371,E2 2561.371} C_VEL
LIN {X 0,Y 562.721,Z 602.81,A -85,B 0,C 180,E1 2568.635,E2 2568.635} C_VEL
LIN {X 0,Y 562.561,Z 602.81,A -85,B 0,C 180,E1 2578.252,E2 2578.252} C_VEL
LIN {X 0,Y 562.309,Z 602.81,A -85,B 0,C 180,E1 2586.952,E2 2586.952} C_VEL
LIN {X 0,Y 562.849,Z 602.81,A -85,B 0,C 180,E1 2595.148,E2 2595.148} C_VEL
LIN {X 0,Y 563.149,Z 602.81,A -85,B 0,C 180,E1 2603.023,E2 2603.023} C_VEL
LIN {X 0,Y 562.949,Z 602.81,A -85,B 0,C 180,E1 2610.76,E2 2610.76} C_VEL
LIN {X 0,Y 562.734,Z 602.81,A -85,B 0,C 180,E1 2618.516,E2 2618.516} C_VEL
LIN {X 0,Y 562.592,Z 602.81,A -85,B 0,C 180,E1 2626.761,E2 2626.761} C_VEL
LIN {X 0,Y 562.593,Z 602.81,A -85,B 0,C 180,E1 2635.369,E2 2635.369} C_VEL
LIN {X 0,Y 562.715,Z 602.81,A -85,B 0,C 180,E1 2644.667,E2 2644.667} C_VEL
LIN {X 0,Y 562.856,Z 602.81,A -85,B 0,C 180,E1 2654.404,E2 2654.404} C_VEL
LIN {X 0,Y 562.544,Z 602.81,A -85,B 0,C 180,E1 2664.553,E2 2664.553} C_VEL
LIN {X 0,Y 562.599,Z 602.81,A -85,B 0,C 180,E1 2673.575,E2 2673.575} C_VEL
LIN {X 0,Y 563.16,Z 604.453,A -85,B 0,C 180,E1 2677.927,E2 2677.927} C_VEL
LIN {X 0,Y 566.577,Z 639.535,A -85,B 0,C 180,E1 2678.896,E2 2678.896} C_VEL
LIN {X 0,Y 565.392,Z 691.223,A -85,B 0,C 180,E1 2681.416,E2 2681.416} C_VEL
LIN {X 0,Y 564.307,Z 734.175,A -85,B 0,C 180,E1 2685.2,E2 2685.2} C_VEL
LIN {X 0,Y 563.371,Z 765.987,A -85,B 0,C 180,E1 2689.918,E2 2689.918} C_VEL
LIN {X 0,Y 563.23,Z 783.338,A -85,B 0,C 180,E1 2694.59,E2 2694.59} C_VEL
LIN {X 0,Y 563.329,Z 789.84,A -85,B 0,C 180,E1 2699.229,E2 2699.229} C_VEL
LIN {X 0,Y 563.465,Z 785.414,A -85,B 0,C 180,E1 2704.415,E2 2704.415} C_VEL
LIN {X 0,Y 563.661,Z 767.462,A -85,B 0,C 180,E1 2709.688,E2 2709.688} C_VEL
LIN {X 0,Y 564.322,Z 734.68,A -85,B 0,C 180,E1 2714.651,E2 2714.651} C_VEL
LIN {X 0,Y 564.462,Z 723.912,A -85,B 0,C 180,E1 2715.811,E2 2715.811} C_VEL
LIN {X 0,Y 557.759,Z 698.409,A -85,B 0,C 180,E1 2718.24,E2 2718.24} C_VEL
LIN {X 0,Y 559.001,Z 648.288,A -85,B 0,C 180,E1 2720.995,E2 2720.995} C_VEL
LIN {X 0,Y 557.311,Z 611.066,A -85,B 0,C 180,E1 2722.117,E2 2722.117} C_VEL
LIN {X 0,Y 554.677,Z 602.81,A -85,B 0,C 180,E1 2722.563,E2 2722.563} C_VEL
LIN {X 0,Y 554.507,Z 602.81,A -85,B 0,C 180,E1 2730.487,E2 2730.487} C_VEL
LIN {X 0,Y 554.506,Z 602.81,A -85,B 0,C 180,E1 2738.771,E2 2738.771} C_VEL
LIN {X 0,Y 554.506,Z 602.81,A -85,B 0,C 180,E1 2746.488,E2 2746.488} C_VEL
LIN {X 0,Y 554.553,Z 602.81,A -85,B 0,C 180,E1 2753.981,E2 2753.981} C_VEL
LIN {X 0,Y 554.767,Z 602.81,A -85,B 0,C 180,E1 2763.187,E2 2763.187} C_VEL
LIN {X 0,Y 555.152,Z 604.662,A -85,B 0,C 180,E1 2766.814,E2 2766.814} C_VEL
LIN {X 0,Y 559.226,Z 626.422,A -85,B 0,C 180,E1 2767.29,E2 2767.29} C_VEL
LIN {X 0,Y 559.027,Z 700.679,A -85,B 0,C 180,E1 2768.679,E2 2768.679} C_VEL
LIN {X 0,Y 557.859,Z 752.245,A -85,B 0,C 180,E1 2771.272,E2 2771.272} C_VEL
LIN {X 0,Y 556.697,Z 795.233,A -85,B 0,C 180,E1 2775.164,E2 2775.164} C_VEL
LIN {X 0,Y 555.746,Z 827.758,A -85,B 0,C 180,E1 2780.188,E2 2780.188} C_VEL
LIN {X 0,Y 555.414,Z 845.075,A -85,B 0,C 180,E1 2785.312,E2 2785.312} C_VEL
LIN {X 0,Y 555.231,Z 849.835,A -85,B 0,C 180,E1 2790.796,E2 2790.796} C_VEL
LIN {X 0,Y 555.245,Z 842.223,A -85,B 0,C 180,E1 2795.895,E2 2795.895} C_VEL
LIN {X 0,Y 555.65,Z 821.149,A -85,B 0,C 180,E1 2801.098,E2 2801.098} C_VEL
LIN {X 0,Y 556.646,Z 786.294,A -85,B 0,C 180,E1 2805.832,E2 2805.832} C_VEL
LIN {X 0,Y 558.165,Z 740.699,A -85,B 0,C 180,E1 2809.465,E2 2809.465} C_VEL
LIN {X 0,Y 559.365,Z 688.556,A -85,B 0,C 180,E1 2811.678,E2 2811.678} C_VEL
LIN {X 0,Y 557.259,Z 610.01,A -85,B 0,C 180,E1 2813.02,E2 2813.02} C_VEL
LIN {X 0,Y 554.995,Z 602.81,A -85,B 0,C 180,E1 2813.369,E2 2813.369} C_VEL
LIN {X 0,Y 554.349,Z 602.81,A -85,B 0,C 180,E1 2822.274,E2 2822.274} C_VEL
LIN {X 0,Y 554.45,Z 602.81,A -85,B 0,C 180,E1 2830.042,E2 2830.042} C_VEL
LIN {X 0,Y 554.348,Z 602.81,A -85,B 0,C 180,E1 2837.88,E2 2837.88} C_VEL
LIN {X 0,Y 554.264,Z 602.81,A -85,B 0,C 180,E1 2845.856,E2 2845.856} C_VEL
LIN {X 0,Y 554.568,Z 602.81,A -85,B 0,C 180,E1 2853.159,E2 2853.159} C_VEL
LIN {X 0,Y 554.647,Z 602.81,A -85,B 0,C 180,E1 2861.66,E2 2861.66} C_VEL
LIN {X 0,Y 555.264,Z 604.267,A -85,B 0,C 180,E1 2866.868,E2 2866.868} C_VEL
LIN {X 0,Y 556.561,Z 643.035,A -85,B 0,C 180,E1 2868.795,E2 2868.795} C_VEL
LIN {X 0,Y 555.796,Z 674.522,A -85,B 0,C 180,E1 2871.955,E2 2871.955} C_VEL
LIN {X 0,Y 555.308,Z 694.422,A -85,B 0,C 180,E1 2876.081,E2 2876.081} C_VEL
LIN {X 0,Y 555.798,Z 699.75,A -85,B 0,C 180,E1 2879.217,E2 2879.217} C_VEL
LIN {X 0,Y 555.61,Z 694.162,A -85,B 0,C 180,E1 2883.914,E2 2883.914} C_VEL
LIN {X 0,Y 555.88,Z 673.897,A -85,B 0,C 180,E1 2888.041,E2 2888.041} C_VEL
LIN {X 0,Y 556.582,Z 641.346,A -85,B 0,C 180,E1 2891.234,E2 2891.234} C_VEL
LIN {X 0,Y 555.644,Z 602.81,A -85,B 0,C 180,E1 2893.221,E2 2893.221} C_VEL
LIN {X 0,Y 554.937,Z 602.81,A -85,B 0,C 180,E1 2903.622,E2 2903.622} C_VEL
LIN {X 0,Y 554.567,Z 602.81,A -85,B 0,C 180,E1 2912.246,E2 2912.246} C_VEL
LIN {X 0,Y 554.499,Z 602.81,A -85,B 0,C 180,E1 2921.171,E2 2921.171} C_VEL
LIN {X 0,Y 554.388,Z 602.81,A -85,B 0,C 180,E1 2929.953,E2 2929.953} C_VEL
LIN {X 0,Y 554.591,Z 602.81,A -85,B 0,C 180,E1 2937.741,E2 2937.741} C_VEL
LIN {X 0,Y 554.366,Z 602.81,A -85,B 0,C 180,E1 2946.603,E2 2946.603} C_VEL
LIN {X 0,Y 554.859,Z 602.81,A -85,B 0,C 180,E1 2954.929,E2 2954.929} C_VEL
LIN {X 0,Y 555.157,Z 602.81,A -85,B 0,C 180,E1 2962.922,E2 2962.922} C_VEL
LIN {X 0,Y 554.944,Z 602.81,A -85,B 0,C 180,E1 2970.771,E2 2970.771} C_VEL
LIN {X 0,Y 554.743,Z 602.81,A -85,B 0,C 180,E1 2978.639,E2 2978.639} C_VEL
LIN {X 0,Y 554.59,Z 602.81,A -85,B 0,C 180,E1 2986.682,E2 2986.682} C_VEL
LIN {X 0,Y 554.567,Z 602.81,A -85,B 0,C 180,E1 2995.079,E2 2995.079} C_VEL
LIN {X 0,Y 554.58,Z 602.81,A -85,B 0,C 180,E1 3004.102,E2 3004.102} C_VEL
LIN {X 0,Y 554.821,Z 602.81,A -85,B 0,C 180,E1 3013.55,E2 3013.55} C_VEL
LIN {X 0,Y 554.579,Z 602.81,A -85,B 0,C 180,E1 3023.965,E2 3023.965} C_VEL
LIN {X 0,Y 554.614,Z 602.81,A -85,B 0,C 180,E1 3033.164,E2 3033.164} C_VEL
LIN {X 0,Y 554.822,Z 602.81,A -85,B 0,C 180,E1 3037.551,E2 3037.551} C_VEL
LIN {X 0,Y 559.168,Z 631.823,A -85,B 0,C 180,E1 3038.36,E2 3038.36} C_VEL
LIN {X 0,Y 557.882,Z 685.029,A -85,B 0,C 180,E1 3040.744,E2 3040.744} C_VEL
LIN {X 0,Y 556.795,Z 728.734,A -85,B 0,C 180,E1 3044.389,E2 3044.389} C_VEL
LIN {X 0,Y 555.803,Z 762.124,A -85,B 0,C 180,E1 3049.038,E2 3049.038} C_VEL
LIN {X 0,Y 555.281,Z 783.337,A -85,B 0,C 180,E1 3054.513,E2 3054.513} C_VEL
LIN {X 0,Y 555.326,Z 789.836,A -85,B 0,C 180,E1 3059.218,E2 3059.218} C_VEL
LIN {X 0,Y 555.3,Z 784.714,A -85,B 0,C 180,E1 3064.822,E2 3064.822} C_VEL
LIN {X 0,Y 555.568,Z 765.532,A -85,B 0,C 180,E1 3070.228,E2 3070.228} C_VEL
LIN {X 0,Y 556.485,Z 733.377,A -85,B 0,C 180,E1 3075.015,E2 3075.015} C_VEL
LIN {X 0,Y 557.759,Z 698.409,A -85,B 0,C 180,E1 3078.24,E2 3078.24} C_VEL
LIN {X 0,Y 550.907,Z 669.963,A -85,B 0,C 180,E1 3080.31,E2 3080.31} C_VEL
LIN {X 0,Y 550.76,Z 615.51,A -85,B 0,C 180,E1 3082.309,E2 3082.309} C_VEL
LIN {X 0,Y 546.648,Z 602.81,A -85,B 0,C 180,E1 3082.872,E2 3082.872} C_VEL
LIN {X 0,Y 546.426,Z 602.81,A -85,B 0,C 180,E1 3090.916,E2 3090.916} C_VEL
LIN {X 0,Y 546.522,Z 602.81,A -85,B 0,C 180,E1 3098.664,E2 3098.664} C_VEL
LIN {X 0,Y 546.342,Z 602.81,A -85,B 0,C 180,E1 3107.397,E2 3107.397} C_VEL
LIN {X 0,Y 546.276,Z 602.81,A -85,B 0,C 180,E1 3115.306,E2 3115.306} C_VEL
LIN {X 0,Y 546.668,Z 602.81,A -85,B 0,C 180,E1 3124.532,E2 3124.532} C_VEL
LIN {X 0,Y 546.983,Z 604.06,A -85,B 0,C 180,E1 3126.439,E2 3126.439} C_VEL
LIN {X 0,Y 551.818,Z 624.219,A -85,B 0,C 180,E1 3126.937,E2 3126.937} C_VEL
LIN {X 0,Y 551.553,Z 699.866,A -85,B 0,C 180,E1 3128.349,E2 3128.349} C_VEL
LIN {X 0,Y 550.271,Z 750.722,A -85,B 0,C 180,E1 3130.9,E2 3130.9} C_VEL
LIN {X 0,Y 548.894,Z 793.866,A -85,B 0,C 180,E1 3134.788,E2 3134.788} C_VEL
LIN {X 0,Y 548.025,Z 825.808,A -85,B 0,C 180,E1 3139.645,E2 3139.645} C_VEL
LIN {X 0,Y 547.435,Z 845.074,A -85,B 0,C 180,E1 3145.243,E2 3145.243} C_VEL
LIN {X 0,Y 547.257,Z 849.834,A -85,B 0,C 180,E1 3150.807,E2 3150.807} C_VEL
LIN {X 0,Y 547.229,Z 842.223,A -85,B 0,C 180,E1 3155.981,E2 3155.981} C_VEL
LIN {X 0,Y 547.686,Z 820.742,A -85,B 0,C 180,E1 3161.337,E2 3161.337} C_VEL
LIN {X 0,Y 548.84,Z 786.293,A -85,B 0,C 180,E1 3166.063,E2 3166.063} C_VEL
LIN {X 0,Y 550.569,Z 740.696,A -85,B 0,C 180,E1 3169.745,E2 3169.745} C_VEL
LIN {X 0,Y 551.941,Z 688.173,A -85,B 0,C 180,E1 3171.995,E2 3171.995} C_VEL
LIN {X 0,Y 549.815,Z 611.777,A -85,B 0,C 180,E1 3173.325,E2 3173.325} C_VEL
LIN {X 0,Y 546.961,Z 602.81,A -85,B 0,C 180,E1 3173.733,E2 3173.733} C_VEL
LIN {X 0,Y 546.374,Z 602.81,A -85,B 0,C 180,E1 3182.804,E2 3182.804} C_VEL
LIN {X 0,Y 546.456,Z 602.81,A -85,B 0,C 180,E1 3190.75,E2 3190.75} C_VEL
LIN {X 0,Y 546.324,Z 602.81,A -85,B 0,C 180,E1 3199.25,E2 3199.25} C_VEL
LIN {X 0,Y 546.267,Z 602.81,A -85,B 0,C 180,E1 3207.932,E2 3207.932} C_VEL
LIN {X 0,Y 546.343,Z 602.81,A -85,B 0,C 180,E1 3216.249,E2 3216.249} C_VEL
LIN {X 0,Y 546.422,Z 602.81,A -85,B 0,C 180,E1 3224.702,E2 3224.702} C_VEL
LIN {X 0,Y 547.177,Z 604.2,A -85,B 0,C 180,E1 3226.671,E2 3226.671} C_VEL
LIN {X 0,Y 548.769,Z 641.006,A -85,B 0,C 180,E1 3228.49,E2 3228.49} C_VEL
LIN {X 0,Y 547.984,Z 673.095,A -85,B 0,C 180,E1 3231.639,E2 3231.639} C_VEL
LIN {X 0,Y 547.583,Z 693.391,A -85,B 0,C 180,E1 3235.678,E2 3235.678} C_VEL
LIN {X 0,Y 547.793,Z 699.74,A -85,B 0,C 180,E1 3239.205,E2 3239.205} C_VEL
LIN {X 0,Y 547.608,Z 694.156,A -85,B 0,C 180,E1 3243.971,E2 3243.971} C_VEL
LIN {X 0,Y 547.915,Z 673.89,A -85,B 0,C 180,E1 3248.159,E2 3248.159} C_VEL
LIN {X 0,Y 548.672,Z 640.944,A -85,B 0,C 180,E1 3251.426,E2 3251.426} C_VEL
LIN {X 0,Y 547.599,Z 602.81,A -85,B 0,C 180,E1 3253.418,E2 3253.418} C_VEL
LIN {X 0,Y 546.92,Z 602.81,A -85,B 0,C 180,E1 3263.722,E2 3263.722} C_VEL
LIN {X 0,Y 546.416,Z 602.81,A -85,B 0,C 180,E1 3272.787,E2 3272.787} C_VEL
LIN {X 0,Y 546.527,Z 602.81,A -85,B 0,C 180,E1 3280.728,E2 3280.728} C_VEL
LIN {X 0,Y 546.425,Z 602.81,A -85,B 0,C 180,E1 3289.79,E2 3289.79} C_VEL
LIN {X 0,Y 546.361,Z 602.81,A -85,B 0,C 180,E1 3299.069,E2 3299.069} C_VEL
LIN {X 0,Y 546.461,Z 602.81,A -85,B 0,C 180,E1 3306.244,E2 3306.244} C_VEL
LIN {X 0,Y 546.862,Z 602.81,A -85,B 0,C 180,E1 3314.703,E2 3314.703} C_VEL
LIN {X 0,Y 547.158,Z 602.81,A -85,B 0,C 180,E1 3322.818,E2 3322.818} C_VEL
LIN {X 0,Y 546.954,Z 602.81,A -85,B 0,C 180,E1 3330.782,E2 3330.782} C_VEL
LIN {X 0,Y 546.726,Z 602.81,A -85,B 0,C 180,E1 3338.767,E2 3338.767} C_VEL
LIN {X 0,Y 546.597,Z 602.81,A -85,B 0,C 180,E1 3346.933,E2 3346.933} C_VEL
LIN {X 0,Y 546.609,Z 602.81,A -85,B 0,C 180,E1 3355.547,E2 3355.547} C_VEL
LIN {X 0,Y 546.634,Z 602.81,A -85,B 0,C 180,E1 3365.024,E2 3365.024} C_VEL
LIN {X 0,Y 546.712,Z 602.81,A -85,B 0,C 180,E1 3375.032,E2 3375.032} C_VEL
LIN {X 0,Y 546.577,Z 602.81,A -85,B 0,C 180,E1 3383.353,E2 3383.353} C_VEL
LIN {X 0,Y 546.682,Z 602.81,A -85,B 0,C 180,E1 3392.743,E2 3392.743} C_VEL
LIN {X 0,Y 546.851,Z 604.018,A -85,B 0,C 180,E1 3397.231,E2 3397.231} C_VEL
LIN {X 0,Y 551.746,Z 629.264,A -85,B 0,C 180,E1 3397.978,E2 3397.978} C_VEL
LIN {X 0,Y 550.397,Z 681.666,A -85,B 0,C 180,E1 3400.262,E2 3400.262} C_VEL
LIN {X 0,Y 549.078,Z 726.836,A -85,B 0,C 180,E1 3403.958,E2 3403.958} C_VEL
LIN {X 0,Y 548.027,Z 761.069,A -85,B 0,C 180,E1 3408.683,E2 3408.683} C_VEL
LIN {X 0,Y 547.493,Z 782.375,A -85,B 0,C 180,E1 3414.035,E2 3414.035} C_VEL
LIN {X 0,Y 547.342,Z 789.833,A -85,B 0,C 180,E1 3419.207,E2 3419.207} C_VEL
LIN {X 0,Y 547.4,Z 785.352,A -85,B 0,C 180,E1 3424.58,E2 3424.58} C_VEL
LIN {X 0,Y 547.673,Z 767.457,A -85,B 0,C 180,E1 3429.974,E2 3429.974} C_VEL
LIN {X 0,Y 548.586,Z 735.207,A -85,B 0,C 180,E1 3435.016,E2 3435.016} C_VEL
LIN {X 0,Y 550.216,Z 691.384,A -85,B 0,C 180,E1 3439.014,E2 3439.014} C_VEL
LIN {X 0,Y 550.907,Z 669.963,A -85,B 0,C 180,E1 3440.31,E2 3440.31} C_VEL
LIN {X 0,Y 544.285,Z 638.821,A -85,B 0,C 180,E1 3441.943,E2 3441.943} C_VEL
LIN {X 0,Y 541.92,Z 613.547,A -85,B 0,C 180,E1 3442.701,E2 3442.701} C_VEL
LIN {X 0,Y 538.603,Z 602.81,A -85,B 0,C 180,E1 3443.104,E2 3443.104} C_VEL
LIN {X 0,Y 538.341,Z 602.81,A -85,B 0,C 180,E1 3451.433,E2 3451.433} C_VEL
LIN {X 0,Y 538.438,Z 602.81,A -85,B 0,C 180,E1 3459.356,E2 3459.356} C_VEL
LIN {X 0,Y 538.244,Z 602.81,A -85,B 0,C 180,E1 3468.528,E2 3468.528} C_VEL
LIN {X 0,Y 538.154,Z 602.81,A -85,B 0,C 180,E1 3476.662,E2 3476.662} C_VEL
LIN {X 0,Y 538.775,Z 602.81,A -85,B 0,C 180,E1 3485.912,E2 3485.912} C_VEL
LIN {X 0,Y 544.47,Z 625.623,A -85,B 0,C 180,E1 3486.631,E2 3486.631} C_VEL
LIN {X 0,Y 544.102,Z 700.392,A -85,B 0,C 180,E1 3488.054,E2 3488.054} C_VEL
LIN {X 0,Y 542.568,Z 752.251,A -85,B 0,C 180,E1 3490.724,E2 3490.724} C_VEL
LIN {X 0,Y 541.034,Z 795.14,A -85,B 0,C 180,E1 3494.713,E2 3494.713} C_VEL
LIN {X 0,Y 540.113,Z 825.807,A -85,B 0,C 180,E1 3499.492,E2 3499.492} C_VEL
LIN {X 0,Y 539.468,Z 845.074,A -85,B 0,C 180,E1 3505.173,E2 3505.173} C_VEL
LIN {X 0,Y 539.253,Z 849.834,A -85,B 0,C 180,E1 3510.819,E2 3510.819} C_VEL
LIN {X 0,Y 539.208,Z 842.224,A -85,B 0,C 180,E1 3516.071,E2 3516.071} C_VEL
LIN {X 0,Y 539.721,Z 820.415,A -85,B 0,C 180,E1 3521.569,E2 3521.569} C_VEL
LIN {X 0,Y 541.014,Z 786.292,A -85,B 0,C 180,E1 3526.302,E2 3526.302} C_VEL
LIN {X 0,Y 542.945,Z 740.692,A -85,B 0,C 180,E1 3530.034,E2 3530.034} C_VEL
LIN {X 0,Y 544.527,Z 688.172,A -85,B 0,C 180,E1 3532.311,E2 3532.311} C_VEL
LIN {X 0,Y 542.456,Z 613.762,A -85,B 0,C 180,E1 3533.599,E2 3533.599} C_VEL
LIN {X 0,Y 538.942,Z 602.81,A -85,B 0,C 180,E1 3533.91,E2 3533.91} C_VEL
LIN {X 0,Y 538.372,Z 602.81,A -85,B 0,C 180,E1 3543.355,E2 3543.355} C_VEL
LIN {X 0,Y 538.474,Z 602.81,A -85,B 0,C 180,E1 3551.684,E2 3551.684} C_VEL
LIN {X 0,Y 538.49,Z 602.81,A -85,B 0,C 180,E1 3560.816,E2 3560.816} C_VEL
LIN {X 0,Y 538.605,Z 602.81,A -85,B 0,C 180,E1 3570.457,E2 3570.457} C_VEL
LIN {X 0,Y 538.717,Z 602.81,A -85,B 0,C 180,E1 3581.098,E2 3581.098} C_VEL
LIN {X 0,Y 539.156,Z 604.617,A -85,B 0,C 180,E1 3586.433,E2 3586.433} C_VEL
LIN {X 0,Y 541.019,Z 639.256,A -85,B 0,C 180,E1 3588.163,E2 3588.163} C_VEL
LIN {X 0,Y 540.147,Z 671.669,A -85,B 0,C 180,E1 3591.314,E2 3591.314} C_VEL
LIN {X 0,Y 539.809,Z 691.927,A -85,B 0,C 180,E1 3595.161,E2 3595.161} C_VEL
LIN {X 0,Y 539.779,Z 699.731,A -85,B 0,C 180,E1 3599.193,E2 3599.193} C_VEL
LIN {X 0,Y 539.603,Z 694.15,A -85,B 0,C 180,E1 3604.03,E2 3604.03} C_VEL
LIN {X 0,Y 539.94,Z 673.883,A -85,B 0,C 180,E1 3608.28,E2 3608.28} C_VEL
LIN {X 0,Y 540.809,Z 641.38,A -85,B 0,C 180,E1 3611.581,E2 3611.581} C_VEL
LIN {X 0,Y 539.599,Z 602.81,A -85,B 0,C 180,E1 3613.621,E2 3613.621} C_VEL
LIN {X 0,Y 538.825,Z 602.81,A -85,B 0,C 180,E1 3624.1,E2 3624.1} C_VEL
LIN {X 0,Y 538.183,Z 602.81,A -85,B 0,C 180,E1 3633.7,E2 3633.7} C_VEL
LIN {X 0,Y 538.342,Z 602.81,A -85,B 0,C 180,E1 3641.656,E2 3641.656} C_VEL
LIN {X 0,Y 538.249,Z 602.81,A -85,B 0,C 180,E1 3650.616,E2 3650.616} C_VEL
LIN {X 0,Y 538.328,Z 602.81,A -85,B 0,C 180,E1 3659.287,E2 3659.287} C_VEL
LIN {X 0,Y 538.1,Z 602.81,A -85,B 0,C 180,E1 3667.61,E2 3667.61} C_VEL
LIN {X 0,Y 538.584,Z 602.81,A -85,B 0,C 180,E1 3676.131,E2 3676.131} C_VEL
LIN {X 0,Y 538.873,Z 602.81,A -85,B 0,C 180,E1 3684.331,E2 3684.331} C_VEL
LIN {X 0,Y 538.797,Z 602.81,A -85,B 0,C 180,E1 3692.408,E2 3692.408} C_VEL
LIN {X 0,Y 538.771,Z 602.81,A -85,B 0,C 180,E1 3700.535,E2 3700.535} C_VEL
LIN {X 0,Y 538.848,Z 602.81,A -85,B 0,C 180,E1 3709.371,E2 3709.371} C_VEL
LIN {X 0,Y 538.675,Z 602.81,A -85,B 0,C 180,E1 3719.519,E2 3719.519} C_VEL
LIN {X 0,Y 538.487,Z 602.81,A -85,B 0,C 180,E1 3729.201,E2 3729.201} C_VEL
LIN {X 0,Y 538.283,Z 602.81,A -85,B 0,C 180,E1 3738.312,E2 3738.312} C_VEL
LIN {X 0,Y 538.159,Z 602.81,A -85,B 0,C 180,E1 3746.645,E2 3746.645} C_VEL
LIN {X 0,Y 538.469,Z 602.81,A -85,B 0,C 180,E1 3754.101,E2 3754.101} C_VEL
LIN {X 0,Y 538.81,Z 604.253,A -85,B 0,C 180,E1 3756.909,E2 3756.909} C_VEL
LIN {X 0,Y 544.27,Z 629.035,A -85,B 0,C 180,E1 3757.659,E2 3757.659} C_VEL
LIN {X 0,Y 542.817,Z 681.658,A -85,B 0,C 180,E1 3759.975,E2 3759.975} C_VEL
LIN {X 0,Y 541.298,Z 726.823,A -85,B 0,C 180,E1 3763.721,E2 3763.721} C_VEL
LIN {X 0,Y 540.046,Z 761.812,A -85,B 0,C 180,E1 3768.658,E2 3768.658} C_VEL
LIN {X 0,Y 539.341,Z 783.329,A -85,B 0,C 180,E1 3774.35,E2 3774.35} C_VEL
LIN {X 0,Y 539.34,Z 789.83,A -85,B 0,C 180,E1 3779.195,E2 3779.195} C_VEL
LIN {X 0,Y 539.298,Z 784.98,A -85,B 0,C 180,E1 3784.844,E2 3784.844} C_VEL
LIN {X 0,Y 539.644,Z 766.098,A -85,B 0,C 180,E1 3790.418,E2 3790.418} C_VEL
LIN {X 0,Y 540.822,Z 733.393,A -85,B 0,C 180,E1 3795.461,E2 3795.461} C_VEL
LIN {X 0,Y 542.624,Z 689.864,A -85,B 0,C 180,E1 3799.397,E2 3799.397} C_VEL
LIN {X 0,Y 544.285,Z 638.821,A -85,B 0,C 180,E1 3801.943,E2 3801.943} C_VEL
LIN {X 0,Y 535.324,Z 618.276,A -85,B 0,C 180,E1 3802.853,E2 3802.853} C_VEL
LIN {X 0,Y 530.534,Z 602.81,A -85,B 0,C 180,E1 3803.514,E2 3803.514} C_VEL
LIN {X 0,Y 530.262,Z 602.81,A -85,B 0,C 180,E1 3812.444,E2 3812.444} C_VEL
LIN {X 0,Y 530.341,Z 602.81,A -85,B 0,C 180,E1 3820.715,E2 3820.715} C_VEL
LIN {X 0,Y 530.274,Z 602.81,A -85,B 0,C 180,E1 3829.94,E2 3829.94} C_VEL
LIN {X 0,Y 530.23,Z 602.81,A -85,B 0,C 180,E1 3838.05,E2 3838.05} C_VEL
LIN {X 0,Y 530.827,Z 603.596,A -85,B 0,C 180,E1 3845.832,E2 3845.832} C_VEL
LIN {X 0,Y 536.958,Z 629.881,A -85,B 0,C 180,E1 3846.421,E2 3846.421} C_VEL
LIN {X 0,Y 536.539,Z 701.035,A -85,B 0,C 180,E1 3847.789,E2 3847.789} C_VEL
LIN {X 0,Y 535.011,Z 750.716,A -85,B 0,C 180,E1 3850.333,E2 3850.333} C_VEL
LIN {X 0,Y 533.257,Z 793.865,A -85,B 0,C 180,E1 3854.331,E2 3854.331} C_VEL
LIN {X 0,Y 532.186,Z 825.807,A -85,B 0,C 180,E1 3859.333,E2 3859.333} C_VEL
LIN {X 0,Y 531.496,Z 845.073,A -85,B 0,C 180,E1 3865.1,E2 3865.1} C_VEL
LIN {X 0,Y 531.262,Z 849.834,A -85,B 0,C 180,E1 3870.832,E2 3870.832} C_VEL
LIN {X 0,Y 531.199,Z 842.224,A -85,B 0,C 180,E1 3876.163,E2 3876.163} C_VEL
LIN {X 0,Y 531.774,Z 821.504,A -85,B 0,C 180,E1 3881.535,E2 3881.535} C_VEL
LIN {X 0,Y 533.185,Z 788.215,A -85,B 0,C 180,E1 3886.335,E2 3886.335} C_VEL
LIN {X 0,Y 535.326,Z 742.479,A -85,B 0,C 180,E1 3890.218,E2 3890.218} C_VEL
LIN {X 0,Y 536.88,Z 691.288,A -85,B 0,C 180,E1 3892.507,E2 3892.507} C_VEL
LIN {X 0,Y 534.714,Z 615.466,A -85,B 0,C 180,E1 3893.823,E2 3893.823} C_VEL
LIN {X 0,Y 530.884,Z 602.81,A -85,B 0,C 180,E1 3894.213,E2 3894.213} C_VEL
LIN {X 0,Y 530.439,Z 602.81,A -85,B 0,C 180,E1 3903.921,E2 3903.921} C_VEL
LIN {X 0,Y 530.517,Z 602.81,A -85,B 0,C 180,E1 3913.162,E2 3913.162} C_VEL
LIN {X 0,Y 530.515,Z 602.81,A -85,B 0,C 180,E1 3922.048,E2 3922.048} C_VEL
LIN {X 0,Y 530.573,Z 602.81,A -85,B 0,C 180,E1 3931.84,E2 3931.84} C_VEL
LIN {X 0,Y 530.742,Z 602.81,A -85,B 0,C 180,E1 3940.802,E2 3940.802} C_VEL
LIN {X 0,Y 531.014,Z 604.538,A -85,B 0,C 180,E1 3946.169,E2 3946.169} C_VEL
LIN {X 0,Y 533.447,Z 634.254,A -85,B 0,C 180,E1 3947.593,E2 3947.593} C_VEL
LIN {X 0,Y 532.532,Z 668.182,A -85,B 0,C 180,E1 3950.595,E2 3950.595} C_VEL
LIN {X 0,Y 531.902,Z 691.015,A -85,B 0,C 180,E1 3954.679,E2 3954.679} C_VEL
LIN {X 0,Y 531.784,Z 700.036,A -85,B 0,C 180,E1 3959.181,E2 3959.181} C_VEL
LIN {X 0,Y 531.605,Z 694.587,A -85,B 0,C 180,E1 3964.091,E2 3964.091} C_VEL
LIN {X 0,Y 532.049,Z 674.668,A -85,B 0,C 180,E1 3968.404,E2 3968.404} C_VEL
LIN {X 0,Y 533.031,Z 642.852,A -85,B 0,C 180,E1 3971.702,E2 3971.702} C_VEL
LIN {X 0,Y 531.794,Z 604.582,A -85,B 0,C 180,E1 3973.667,E2 3973.667} C_VEL
LIN {X 0,Y 530.713,Z 602.81,A -85,B 0,C 180,E1 3984.493,E2 3984.493} C_VEL
LIN {X 0,Y 530.166,Z 602.81,A -85,B 0,C 180,E1 3993.926,E2 3993.926} C_VEL
LIN {X 0,Y 530.229,Z 602.81,A -85,B 0,C 180,E1 4003.116,E2 4003.116} C_VEL
LIN {X 0,Y 530.053,Z 602.81,A -85,B 0,C 180,E1 4011.997,E2 4011.997} C_VEL
LIN {X 0,Y 530.27,Z 602.81,A -85,B 0,C 180,E1 4020.785,E2 4020.785} C_VEL
LIN {X 0,Y 529.994,Z 602.81,A -85,B 0,C 180,E1 4029.016,E2 4029.016} C_VEL
LIN {X 0,Y 530.595,Z 602.81,A -85,B 0,C 180,E1 4035.918,E2 4035.918} C_VEL
LIN {X 0,Y 530.878,Z 602.81,A -85,B 0,C 180,E1 4044.245,E2 4044.245} C_VEL
LIN {X 0,Y 530.989,Z 602.81,A -85,B 0,C 180,E1 4050.805,E2 4050.805} C_VEL
LIN {X 0,Y 530.695,Z 602.81,A -85,B 0,C 180,E1 4059.434,E2 4059.434} C_VEL
LIN {X 0,Y 530.609,Z 602.81,A -85,B 0,C 180,E1 4067.459,E2 4067.459} C_VEL
LIN {X 0,Y 530.676,Z 602.81,A -85,B 0,C 180,E1 4076.293,E2 4076.293} C_VEL
LIN {X 0,Y 530.681,Z 602.81,A -85,B 0,C 180,E1 4085.868,E2 4085.868} C_VEL
LIN {X 0,Y 530.476,Z 602.81,A -85,B 0,C 180,E1 4095.507,E2 4095.507} C_VEL
LIN {X 0,Y 530.391,Z 602.81,A -85,B 0,C 180,E1 4104.598,E2 4104.598} C_VEL
LIN {X 0,Y 530.452,Z 602.81,A -85,B 0,C 180,E1 4114.267,E2 4114.267} C_VEL
LIN {X 0,Y 530.632,Z 603.823,A -85,B 0,C 180,E1 4116.561,E2 4116.561} C_VEL
LIN {X 0,Y 536.765,Z 630.22,A -85,B 0,C 180,E1 4117.395,E2 4117.395} C_VEL
LIN {X 0,Y 535.166,Z 683.243,A -85,B 0,C 180,E1 4119.784,E2 4119.784} C_VEL
LIN {X 0,Y 533.41,Z 728.696,A -85,B 0,C 180,E1 4123.686,E2 4123.686} C_VEL
LIN {X 0,Y 532.052,Z 762.871,A -85,B 0,C 180,E1 4128.693,E2 4128.693} C_VEL
LIN {X 0,Y 531.373,Z 783.325,A -85,B 0,C 180,E1 4134.265,E2 4134.265} C_VEL
LIN {X 0,Y 531.341,Z 789.827,A -85,B 0,C 180,E1 4139.183,E2 4139.183} C_VEL
LIN {X 0,Y 531.279,Z 784.982,A -85,B 0,C 180,E1 4144.917,E2 4144.917} C_VEL
LIN {X 0,Y 531.703,Z 767.129,A -85,B 0,C 180,E1 4150.348,E2 4150.348} C_VEL
LIN {X 0,Y 532.963,Z 735.265,A -85,B 0,C 180,E1 4155.459,E2 4155.459} C_VEL
LIN {X 0,Y 534.953,Z 691.353,A -85,B 0,C 180,E1 4159.579,E2 4159.579} C_VEL
LIN {X 0,Y 536.697,Z 640.087,A -85,B 0,C 180,E1 4162.182,E2 4162.182} C_VEL
LIN {X 0,Y 535.324,Z 618.276,A -85,B 0,C 180,E1 4162.853,E2 4162.853} C_VEL
LIN {X 0,Y 524.235,Z 609.304,A -85,B 0,C 180,E1 4163.462,E2 4163.462} C_VEL
LIN {X 0,Y 522.485,Z 602.81,A -85,B 0,C 180,E1 4163.857,E2 4163.857} C_VEL
LIN {X 0,Y 522.261,Z 602.81,A -85,B 0,C 180,E1 4172.517,E2 4172.517} C_VEL
LIN {X 0,Y 522.343,Z 602.81,A -85,B 0,C 180,E1 4180.819,E2 4180.819} C_VEL
LIN {X 0,Y 522.273,Z 602.81,A -85,B 0,C 180,E1 4190.353,E2 4190.353} C_VEL
LIN {X 0,Y 522.422,Z 602.81,A -85,B 0,C 180,E1 4199.466,E2 4199.466} C_VEL
LIN {X 0,Y 522.797,Z 603.86,A -85,B 0,C 180,E1 4205.529,E2 4205.529} C_VEL
LIN {X 0,Y 529.398,Z 631.276,A -85,B 0,C 180,E1 4206.166,E2 4206.166} C_VEL
LIN {X 0,Y 528.837,Z 701.355,A -85,B 0,C 180,E1 4207.559,E2 4207.559} C_VEL
LIN {X 0,Y 527.18,Z 753.479,A -85,B 0,C 180,E1 4210.282,E2 4210.282} C_VEL
LIN {X 0,Y 525.439,Z 793.864,A -85,B 0,C 180,E1 4214.091,E2 4214.091} C_VEL
LIN {X 0,Y 524.225,Z 825.806,A -85,B 0,C 180,E1 4219.169,E2 4219.169} C_VEL
LIN {X 0,Y 523.539,Z 845.073,A -85,B 0,C 180,E1 4225.026,E2 4225.026} C_VEL
LIN {X 0,Y 523.26,Z 849.833,A -85,B 0,C 180,E1 4230.844,E2 4230.844} C_VEL
LIN {X 0,Y 523.213,Z 842.224,A -85,B 0,C 180,E1 4236.257,E2 4236.257} C_VEL
LIN {X 0,Y 523.799,Z 821.503,A -85,B 0,C 180,E1 4241.713,E2 4241.713} C_VEL
LIN {X 0,Y 525.365,Z 788.213,A -85,B 0,C 180,E1 4246.585,E2 4246.585} C_VEL
LIN {X 0,Y 527.489,Z 744.88,A -85,B 0,C 180,E1 4250.29,E2 4250.29} C_VEL
LIN {X 0,Y 529.175,Z 691.119,A -85,B 0,C 180,E1 4252.733,E2 4252.733} C_VEL
LIN {X 0,Y 527.114,Z 617.405,A -85,B 0,C 180,E1 4254.046,E2 4254.046} C_VEL
LIN {X 0,Y 522.86,Z 602.81,A -85,B 0,C 180,E1 4254.454,E2 4254.454} C_VEL
LIN {X 0,Y 522.478,Z 602.81,A -85,B 0,C 180,E1 4264.51,E2 4264.51} C_VEL
LIN {X 0,Y 522.543,Z 602.81,A -85,B 0,C 180,E1 4274.642,E2 4274.642} C_VEL
LIN {X 0,Y 522.394,Z 602.81,A -85,B 0,C 180,E1 4283.451,E2 4283.451} C_VEL
LIN {X 0,Y 522.397,Z 602.81,A -85,B 0,C 180,E1 4293.239,E2 4293.239} C_VEL
LIN {X 0,Y 522.454,Z 602.81,A -85,B 0,C 180,E1 4302.242,E2 4302.242} C_VEL
LIN {X 0,Y 522.85,Z 604.083,A -85,B 0,C 180,E1 4305.884,E2 4305.884} C_VEL
LIN {X 0,Y 525.817,Z 632.903,A -85,B 0,C 180,E1 4307.249,E2 4307.249} C_VEL
LIN {X 0,Y 524.771,Z 667.537,A -85,B 0,C 180,E1 4310.222,E2 4310.222} C_VEL
LIN {X 0,Y 523.95,Z 690.765,A -85,B 0,C 180,E1 4314.181,E2 4314.181} C_VEL
LIN {X 0,Y 523.74,Z 701.06,A -85,B 0,C 180,E1 4318.733,E2 4318.733} C_VEL
LIN {X 0,Y 523.795,Z 696.812,A -85,B 0,C 180,E1 4323.736,E2 4323.736} C_VEL
LIN {X 0,Y 524.249,Z 678.339,A -85,B 0,C 180,E1 4328.111,E2 4328.111} C_VEL
LIN {X 0,Y 525.223,Z 647.809,A -85,B 0,C 180,E1 4331.561,E2 4331.561} C_VEL
LIN {X 0,Y 524.495,Z 607.764,A -85,B 0,C 180,E1 4333.787,E2 4333.787} C_VEL
LIN {X 0,Y 523.456,Z 602.81,A -85,B 0,C 180,E1 4334.264,E2 4334.264} C_VEL
LIN {X 0,Y 522.637,Z 602.81,A -85,B 0,C 180,E1 4344.897,E2 4344.897} C_VEL
LIN {X 0,Y 522.139,Z 602.81,A -85,B 0,C 180,E1 4354.52,E2 4354.52} C_VEL
LIN {X 0,Y 522.228,Z 602.81,A -85,B 0,C 180,E1 4363.066,E2 4363.066} C_VEL
LIN {X 0,Y 522.071,Z 602.81,A -85,B 0,C 180,E1 4371.309,E2 4371.309} C_VEL
LIN {X 0,Y 522.256,Z 602.81,A -85,B 0,C 180,E1 4379.424,E2 4379.424} C_VEL
LIN {X 0,Y 522.197,Z 602.81,A -85,B 0,C 180,E1 4386.889,E2 4386.889} C_VEL
LIN {X 0,Y 522.613,Z 602.81,A -85,B 0,C 180,E1 4395.698,E2 4395.698} C_VEL
LIN {X 0,Y 522.896,Z 602.81,A -85,B 0,C 180,E1 4404.157,E2 4404.157} C_VEL
LIN {X 0,Y 522.987,Z 602.81,A -85,B 0,C 180,E1 4410.818,E2 4410.818} C_VEL
LIN {X 0,Y 522.715,Z 602.81,A -85,B 0,C 180,E1 4419.173,E2 4419.173} C_VEL
LIN {X 0,Y 522.618,Z 602.81,A -85,B 0,C 180,E1 4427.735,E2 4427.735} C_VEL
LIN {X 0,Y 522.677,Z 602.81,A -85,B 0,C 180,E1 4437.69,E2 4437.69} C_VEL
LIN {X 0,Y 522.543,Z 602.81,A -85,B 0,C 180,E1 4447.005,E2 4447.005} C_VEL
LIN {X 0,Y 522.325,Z 602.81,A -85,B 0,C 180,E1 4456.944,E2 4456.944} C_VEL
LIN {X 0,Y 522.222,Z 602.81,A -85,B 0,C 180,E1 4465.879,E2 4465.879} C_VEL
LIN {X 0,Y 522.4,Z 602.81,A -85,B 0,C 180,E1 4475.091,E2 4475.091} C_VEL
LIN {X 0,Y 522.657,Z 604.164,A -85,B 0,C 180,E1 4476.222,E2 4476.222} C_VEL
LIN {X 0,Y 529.278,Z 632.104,A -85,B 0,C 180,E1 4477.143,E2 4477.143} C_VEL
LIN {X 0,Y 527.525,Z 683.798,A -85,B 0,C 180,E1 4479.532,E2 4479.532} C_VEL
LIN {X 0,Y 525.654,Z 728.705,A -85,B 0,C 180,E1 4483.438,E2 4483.438} C_VEL
LIN {X 0,Y 524.153,Z 762.863,A -85,B 0,C 180,E1 4488.521,E2 4488.521} C_VEL
LIN {X 0,Y 523.435,Z 783.32,A -85,B 0,C 180,E1 4494.178,E2 4494.178} C_VEL
LIN {X 0,Y 523.355,Z 789.824,A -85,B 0,C 180,E1 4499.171,E2 4499.171} C_VEL
LIN {X 0,Y 523.258,Z 784.984,A -85,B 0,C 180,E1 4504.992,E2 4504.992} C_VEL
LIN {X 0,Y 523.714,Z 766.767,A -85,B 0,C 180,E1 4510.589,E2 4510.589} C_VEL
LIN {X 0,Y 525.138,Z 734.996,A -85,B 0,C 180,E1 4515.732,E2 4515.732} C_VEL
LIN {X 0,Y 527.233,Z 692.784,A -85,B 0,C 180,E1 4519.752,E2 4519.752} C_VEL
LIN {X 0,Y 529.124,Z 641.484,A -85,B 0,C 180,E1 4522.422,E2 4522.422} C_VEL
LIN {X 0,Y 526.724,Z 617.065,A -85,B 0,C 180,E1 4523.216,E2 4523.216} C_VEL
LIN {X 0,Y 524.235,Z 609.304,A -85,B 0,C 180,E1 4523.462,E2 4523.462} C_VEL
LIN {X 0,Y 518.744,Z 602.188,A -85,B 0,C 180,E1 4524.681,E2 4524.681} C_VEL
LIN {X 0,Y 514.576,Z 602.81,A -85,B 0,C 180,E1 4527.103,E2 4527.103} C_VEL
LIN {X 0,Y 514.468,Z 602.81,A -85,B 0,C 180,E1 4537.207,E2 4537.207} C_VEL
LIN {X 0,Y 514.339,Z 602.81,A -85,B 0,C 180,E1 4546.291,E2 4546.291} C_VEL
LIN {X 0,Y 514.218,Z 602.81,A -85,B 0,C 180,E1 4554.889,E2 4554.889} C_VEL
LIN {X 0,Y 514.666,Z 602.81,A -85,B 0,C 180,E1 4564.974,E2 4564.974} C_VEL
LIN {X 0,Y 521.83,Z 631.088,A -85,B 0,C 180,E1 4565.88,E2 4565.88} C_VEL
LIN {X 0,Y 521.262,Z 700.252,A -85,B 0,C 180,E1 4567.271,E2 4567.271} C_VEL
LIN {X 0,Y 519.399,Z 752.314,A -85,B 0,C 180,E1 4570.013,E2 4570.013} C_VEL
LIN {X 0,Y 517.45,Z 797.086,A -85,B 0,C 180,E1 4574.276,E2 4574.276} C_VEL
LIN {X 0,Y 516.178,Z 827.53,A -85,B 0,C 180,E1 4579.378,E2 4579.378} C_VEL
LIN {X 0,Y 515.585,Z 845.072,A -85,B 0,C 180,E1 4584.949,E2 4584.949} C_VEL
LIN {X 0,Y 515.256,Z 849.833,A -85,B 0,C 180,E1 4590.857,E2 4590.857} C_VEL
LIN {X 0,Y 515.23,Z 842.224,A -85,B 0,C 180,E1 4596.354,E2 4596.354} C_VEL
LIN {X 0,Y 515.862,Z 821.503,A -85,B 0,C 180,E1 4601.896,E2 4601.896} C_VEL
LIN {X 0,Y 517.456,Z 789.833,A -85,B 0,C 180,E1 4606.584,E2 4606.584} C_VEL
LIN {X 0,Y 519.671,Z 743.946,A -85,B 0,C 180,E1 4610.516,E2 4610.516} C_VEL
LIN {X 0,Y 521.48,Z 690.651,A -85,B 0,C 180,E1 4612.974,E2 4612.974} C_VEL
LIN {X 0,Y 519.565,Z 619.413,A -85,B 0,C 180,E1 4614.273,E2 4614.273} C_VEL
LIN {X 0,Y 514.842,Z 602.81,A -85,B 0,C 180,E1 4614.763,E2 4614.763} C_VEL
LIN {X 0,Y 514.431,Z 602.81,A -85,B 0,C 180,E1 4625.128,E2 4625.128} C_VEL
LIN {X 0,Y 514.476,Z 602.81,A -85,B 0,C 180,E1 4633.895,E2 4633.895} C_VEL
LIN {X 0,Y 514.266,Z 602.81,A -85,B 0,C 180,E1 4644.256,E2 4644.256} C_VEL
LIN {X 0,Y 514.294,Z 602.81,A -85,B 0,C 180,E1 4654.172,E2 4654.172} C_VEL
LIN {X 0,Y 514.352,Z 602.81,A -85,B 0,C 180,E1 4663.537,E2 4663.537} C_VEL
LIN {X 0,Y 514.715,Z 603.782,A -85,B 0,C 180,E1 4665.601,E2 4665.601} C_VEL
LIN {X 0,Y 518.1,Z 633.019,A -85,B 0,C 180,E1 4666.993,E2 4666.993} C_VEL
LIN {X 0,Y 516.97,Z 668.667,A -85,B 0,C 180,E1 4670.069,E2 4670.069} C_VEL
LIN {X 0,Y 516.084,Z 691.971,A -85,B 0,C 180,E1 4674.092,E2 4674.092} C_VEL
LIN {X 0,Y 515.511,Z 700.938,A -85,B 0,C 180,E1 4677.468,E2 4677.468} C_VEL
LIN {X 0,Y 515.724,Z 700.532,A -85,B 0,C 180,E1 4682.528,E2 4682.528} C_VEL
LIN {X 0,Y 516.22,Z 685.263,A -85,B 0,C 180,E1 4687.176,E2 4687.176} C_VEL
LIN {X 0,Y 517.145,Z 657.016,A -85,B 0,C 180,E1 4690.994,E2 4690.994} C_VEL
LIN {X 0,Y 518.072,Z 618.864,A -85,B 0,C 180,E1 4693.554,E2 4693.554} C_VEL
LIN {X 0,Y 515.44,Z 602.81,A -85,B 0,C 180,E1 4694.311,E2 4694.311} C_VEL
LIN {X 0,Y 514.542,Z 602.81,A -85,B 0,C 180,E1 4705.316,E2 4705.316} C_VEL
LIN {X 0,Y 514.236,Z 602.81,A -85,B 0,C 180,E1 4713.086,E2 4713.086} C_VEL
LIN {X 0,Y 514.257,Z 602.81,A -85,B 0,C 180,E1 4721.599,E2 4721.599} C_VEL
LIN {X 0,Y 514.142,Z 602.81,A -85,B 0,C 180,E1 4730.598,E2 4730.598} C_VEL
LIN {X 0,Y 514.217,Z 602.81,A -85,B 0,C 180,E1 4740.521,E2 4740.521} C_VEL
LIN {X 0,Y 514.022,Z 602.81,A -85,B 0,C 180,E1 4748.42,E2 4748.42} C_VEL
LIN {X 0,Y 514.455,Z 602.81,A -85,B 0,C 180,E1 4757.206,E2 4757.206} C_VEL
LIN {X 0,Y 514.802,Z 602.81,A -85,B 0,C 180,E1 4765.76,E2 4765.76} C_VEL
LIN {X 0,Y 514.991,Z 602.81,A -85,B 0,C 180,E1 4774.21,E2 4774.21} C_VEL
LIN {X 0,Y 514.856,Z 602.81,A -85,B 0,C 180,E1 4784.493,E2 4784.493} C_VEL
LIN {X 0,Y 514.558,Z 602.81,A -85,B 0,C 180,E1 4793.444,E2 4793.444} C_VEL
LIN {X 0,Y 514.329,Z 602.81,A -85,B 0,C 180,E1 4803.062,E2 4803.062} C_VEL
LIN {X 0,Y 514.402,Z 602.81,A -85,B 0,C 180,E1 4811.564,E2 4811.564} C_VEL
LIN {X 0,Y 514.426,Z 602.81,A -85,B 0,C 180,E1 4821.39,E2 4821.39} C_VEL
LIN {X 0,Y 514.465,Z 602.81,A -85,B 0,C 180,E1 4830.878,E2 4830.878} C_VEL
LIN {X 0,Y 514.576,Z 603.912,A -85,B 0,C 180,E1 4835.859,E2 4835.859} C_VEL
LIN {X 0,Y 521.793,Z 633.992,A -85,B 0,C 180,E1 4836.885,E2 4836.885} C_VEL
LIN {X 0,Y 519.846,Z 685.685,A -85,B 0,C 180,E1 4839.36,E2 4839.36} C_VEL
LIN {X 0,Y 517.775,Z 730.665,A -85,B 0,C 180,E1 4843.398,E2 4843.398} C_VEL
LIN {X 0,Y 516.147,Z 763.931,A -85,B 0,C 180,E1 4848.555,E2 4848.555} C_VEL
LIN {X 0,Y 515.47,Z 783.316,A -85,B 0,C 180,E1 4854.087,E2 4854.087} C_VEL
LIN {X 0,Y 515.353,Z 789.821,A -85,B 0,C 180,E1 4859.158,E2 4859.158} C_VEL
LIN {X 0,Y 515.238,Z 784.984,A -85,B 0,C 180,E1 4865.07,E2 4865.07} C_VEL
LIN {X 0,Y 515.754,Z 767.006,A -85,B 0,C 180,E1 4870.699,E2 4870.699} C_VEL
LIN {X 0,Y 517.337,Z 735.27,A -85,B 0,C 180,E1 4875.963,E2 4875.963} C_VEL
LIN {X 0,Y 519.613,Z 691.861,A -85,B 0,C 180,E1 4880.099,E2 4880.099} C_VEL
LIN {X 0,Y 521.58,Z 641.22,A -85,B 0,C 180,E1 4882.727,E2 4882.727} C_VEL
LIN {X 0,Y 518.689,Z 617.54,A -85,B 0,C 180,E1 4883.526,E2 4883.526} C_VEL
LIN {X 0,Y 514.477,Z 602.81,A -85,B 0,C 180,E1 4884.102,E2 4884.102} C_VEL
LIN {X 0,Y 514.576,Z 602.81,A -85,B 0,C 180,E1 4887.103,E2 4887.103} C_VEL
LIN {X 0,Y 506.272,Z 602.81,A -85,B 0,C 180,E1 4890.995,E2 4890.995} C_VEL
LIN {X 0,Y 506.291,Z 602.81,A -85,B 0,C 180,E1 4900.183,E2 4900.183} C_VEL
LIN {X 0,Y 506.178,Z 602.81,A -85,B 0,C 180,E1 4909.89,E2 4909.89} C_VEL
LIN {X 0,Y 506.276,Z 602.81,A -85,B 0,C 180,E1 4918.678,E2 4918.678} C_VEL
LIN {X 0,Y 506.743,Z 603.987,A -85,B 0,C 180,E1 4924.887,E2 4924.887} C_VEL
LIN {X 0,Y 514.302,Z 635.442,A -85,B 0,C 180,E1 4925.655,E2 4925.655} C_VEL
LIN {X 0,Y 513.502,Z 702.008,A -85,B 0,C 180,E1 4927.08,E2 4927.08} C_VEL
LIN {X 0,Y 511.52,Z 753.632,A -85,B 0,C 180,E1 4929.926,E2 4929.926} C_VEL
LIN {X 0,Y 509.477,Z 797.423,A -85,B 0,C 180,E1 4934.245,E2 4934.245} C_VEL
LIN {X 0,Y 508.153,Z 828.624,A -85,B 0,C 180,E1 4939.467,E2 4939.467} C_VEL
LIN {X 0,Y 507.616,Z 845.072,A -85,B 0,C 180,E1 4944.869,E2 4944.869} C_VEL
LIN {X 0,Y 507.257,Z 849.833,A -85,B 0,C 180,E1 4950.871,E2 4950.871} C_VEL
LIN {X 0,Y 507.24,Z 842.224,A -85,B 0,C 180,E1 4956.455,E2 4956.455} C_VEL
LIN {X 0,Y 507.891,Z 822.248,A -85,B 0,C 180,E1 4961.867,E2 4961.867} C_VEL
LIN {X 0,Y 509.483,Z 788.393,A -85,B 0,C 180,E1 4966.817,E2 4966.817} C_VEL
LIN {X 0,Y 511.907,Z 741.525,A -85,B 0,C 180,E1 4970.847,E2 4970.847} C_VEL
LIN {X 0,Y 513.793,Z 688.281,A -85,B 0,C 180,E1 4973.281,E2 4973.281} C_VEL
LIN {X 0,Y 511.981,Z 621.093,A -85,B 0,C 180,E1 4974.564,E2 4974.564} C_VEL
LIN {X 0,Y 506.793,Z 602.81,A -85,B 0,C 180,E1 4975.214,E2 4975.214} C_VEL
LIN {X 0,Y 506.463,Z 602.81,A -85,B 0,C 180,E1 4985.765,E2 4985.765} C_VEL
LIN {X 0,Y 506.342,Z 602.81,A -85,B 0,C 180,E1 4995.227,E2 4995.227} C_VEL
LIN {X 0,Y 506.291,Z 602.81,A -85,B 0,C 180,E1 5004.233,E2 5004.233} C_VEL
LIN {X 0,Y 506.298,Z 602.81,A -85,B 0,C 180,E1 5014.239,E2 5014.239} C_VEL
LIN {X 0,Y 506.364,Z 602.81,A -85,B 0,C 180,E1 5023.458,E2 5023.458} C_VEL
LIN {X 0,Y 506.682,Z 604.132,A -85,B 0,C 180,E1 5025.326,E2 5025.326} C_VEL
LIN {X 0,Y 510.452,Z 631.982,A -85,B 0,C 180,E1 5026.665,E2 5026.665} C_VEL
LIN {X 0,Y 509.204,Z 668.094,A -85,B 0,C 180,E1 5029.699,E2 5029.699} C_VEL
LIN {X 0,Y 508.1,Z 691.508,A -85,B 0,C 180,E1 5033.568,E2 5033.568} C_VEL
LIN {X 0,Y 507.629,Z 702.142,A -85,B 0,C 180,E1 5037.429,E2 5037.429} C_VEL
LIN {X 0,Y 507.822,Z 701.656,A -85,B 0,C 180,E1 5042.568,E2 5042.568} C_VEL
LIN {X 0,Y 508.35,Z 686.233,A -85,B 0,C 180,E1 5047.287,E2 5047.287} C_VEL
LIN {X 0,Y 509.347,Z 657.836,A -85,B 0,C 180,E1 5051.165,E2 5051.165} C_VEL
LIN {X 0,Y 510.371,Z 618.448,A -85,B 0,C 180,E1 5053.815,E2 5053.815} C_VEL
LIN {X 0,Y 507.333,Z 602.81,A -85,B 0,C 180,E1 5054.727,E2 5054.727} C_VEL
LIN {X 0,Y 506.653,Z 602.81,A -85,B 0,C 180,E1 5063.981,E2 5063.981} C_VEL
LIN {X 0,Y 506.118,Z 602.81,A -85,B 0,C 180,E1 5073.687,E2 5073.687} C_VEL
LIN {X 0,Y 506.162,Z 602.81,A -85,B 0,C 180,E1 5082.718,E2 5082.718} C_VEL
LIN {X 0,Y 506.032,Z 602.81,A -85,B 0,C 180,E1 5092.052,E2 5092.052} C_VEL
LIN {X 0,Y 506.234,Z 602.81,A -85,B 0,C 180,E1 5100.343,E2 5100.343} C_VEL
LIN {X 0,Y 506.069,Z 602.81,A -85,B 0,C 180,E1 5109.815,E2 5109.815} C_VEL
LIN {X 0,Y 506.557,Z 602.81,A -85,B 0,C 180,E1 5118.758,E2 5118.758} C_VEL
LIN {X 0,Y 507.151,Z 602.81,A -85,B 0,C 180,E1 5127.414,E2 5127.414} C_VEL
LIN {X 0,Y 506.924,Z 602.81,A -85,B 0,C 180,E1 5137.727,E2 5137.727} C_VEL
LIN {X 0,Y 506.582,Z 602.81,A -85,B 0,C 180,E1 5146.517,E2 5146.517} C_VEL
LIN {X 0,Y 506.513,Z 602.81,A -85,B 0,C 180,E1 5155.73,E2 5155.73} C_VEL
LIN {X 0,Y 506.47,Z 602.81,A -85,B 0,C 180,E1 5165.73,E2 5165.73} C_VEL
LIN {X 0,Y 506.317,Z 602.81,A -85,B 0,C 180,E1 5175.228,E2 5175.228} C_VEL
LIN {X 0,Y 506.274,Z 602.81,A -85,B 0,C 180,E1 5184.235,E2 5184.235} C_VEL
LIN {X 0,Y 506.374,Z 602.81,A -85,B 0,C 180,E1 5194.246,E2 5194.246} C_VEL
LIN {X 0,Y 506.485,Z 603.739,A -85,B 0,C 180,E1 5195.484,E2 5195.484} C_VEL
LIN {X 0,Y 514.316,Z 635.541,A -85,B 0,C 180,E1 5196.608,E2 5196.608} C_VEL
LIN {X 0,Y 512.109,Z 688.01,A -85,B 0,C 180,E1 5199.212,E2 5199.212} C_VEL
LIN {X 0,Y 509.884,Z 732.656,A -85,B 0,C 180,E1 5203.365,E2 5203.365} C_VEL
LIN {X 0,Y 508.151,Z 765.266,A -85,B 0,C 180,E1 5208.591,E2 5208.591} C_VEL
LIN {X 0,Y 507.506,Z 783.403,A -85,B 0,C 180,E1 5213.994,E2 5213.994} C_VEL
LIN {X 0,Y 507.352,Z 789.818,A -85,B 0,C 180,E1 5219.144,E2 5219.144} C_VEL
LIN {X 0,Y 507.234,Z 785.067,A -85,B 0,C 180,E1 5225.151,E2 5225.151} C_VEL
LIN {X 0,Y 507.82,Z 767.172,A -85,B 0,C 180,E1 5230.914,E2 5230.914} C_VEL
LIN {X 0,Y 509.525,Z 735.39,A -85,B 0,C 180,E1 5236.214,E2 5236.214} C_VEL
LIN {X 0,Y 511.951,Z 692.52,A -85,B 0,C 180,E1 5240.342,E2 5240.342} C_VEL
LIN {X 0,Y 514.04,Z 641.462,A -85,B 0,C 180,E1 5243.021,E2 5243.021} C_VEL
LIN {X 0,Y 511.04,Z 618.757,A -85,B 0,C 180,E1 5243.814,E2 5243.814} C_VEL
LIN {X 0,Y 506.447,Z 602.81,A -85,B 0,C 180,E1 5244.499,E2 5244.499} C_VEL
LIN {X 0,Y 506.272,Z 602.81,A -85,B 0,C 180,E1 5250.995,E2 5250.995} C_VEL
LIN {X 0,Y 498.26,Z 602.81,A -85,B 0,C 180,E1 5254.948,E2 5254.948} C_VEL
LIN {X 0,Y 498.264,Z 602.81,A -85,B 0,C 180,E1 5264.324,E2 5264.324} C_VEL
LIN {X 0,Y 498.258,Z 602.81,A -85,B 0,C 180,E1 5273.813,E2 5273.813} C_VEL
LIN {X 0,Y 498.611,Z 602.81,A -85,B 0,C 180,E1 5284.24,E2 5284.24} C_VEL
LIN {X 0,Y 500.528,Z 609.835,A -85,B 0,C 180,E1 5284.716,E2 5284.716} C_VEL
LIN {X 0,Y 506.809,Z 637.649,A -85,B 0,C 180,E1 5285.392,E2 5285.392} C_VEL
LIN {X 0,Y 505.836,Z 702.308,A -85,B 0,C 180,E1 5286.83,E2 5286.83} C_VEL
LIN {X 0,Y 503.667,Z 753.788,A -85,B 0,C 180,E1 5289.745,E2 5289.745} C_VEL
LIN {X 0,Y 501.491,Z 797.751,A -85,B 0,C 180,E1 5294.213,E2 5294.213} C_VEL
LIN {X 0,Y 500.15,Z 828.495,A -85,B 0,C 180,E1 5299.526,E2 5299.526} C_VEL
LIN {X 0,Y 499.302,Z 846.42,A -85,B 0,C 180,E1 5305.657,E2 5305.657} C_VEL
LIN {X 0,Y 499.254,Z 849.762,A -85,B 0,C 180,E1 5310.885,E2 5310.885} C_VEL
LIN {X 0,Y 499.225,Z 841.752,A -85,B 0,C 180,E1 5316.559,E2 5316.559} C_VEL
LIN {X 0,Y 499.957,Z 820.832,A -85,B 0,C 180,E1 5322.058,E2 5322.058} C_VEL
LIN {X 0,Y 501.609,Z 786.517,A -85,B 0,C 180,E1 5327.103,E2 5327.103} C_VEL
LIN {X 0,Y 504.126,Z 739.273,A -85,B 0,C 180,E1 5331.184,E2 5331.184} C_VEL
LIN {X 0,Y 506.3,Z 685.588,A -85,B 0,C 180,E1 5333.646,E2 5333.646} C_VEL
LIN {X 0,Y 504.501,Z 622.537,A -85,B 0,C 180,E1 5334.893,E2 5334.893} C_VEL
LIN {X 0,Y 498.767,Z 602.81,A -85,B 0,C 180,E1 5335.57,E2 5335.57} C_VEL
LIN {X 0,Y 498.432,Z 602.81,A -85,B 0,C 180,E1 5346.214,E2 5346.214} C_VEL
LIN {X 0,Y 498.258,Z 602.81,A -85,B 0,C 180,E1 5355.717,E2 5355.717} C_VEL
LIN {X 0,Y 498.156,Z 602.81,A -85,B 0,C 180,E1 5365.697,E2 5365.697} C_VEL
LIN {X 0,Y 498.291,Z 602.81,A -85,B 0,C 180,E1 5373.969,E2 5373.969} C_VEL
LIN {X 0,Y 498.378,Z 602.81,A -85,B 0,C 180,E1 5383.596,E2 5383.596} C_VEL
LIN {X 0,Y 498.654,Z 604.314,A -85,B 0,C 180,E1 5385.032,E2 5385.032} C_VEL
LIN {X 0,Y 502.752,Z 633.207,A -85,B 0,C 180,E1 5386.457,E2 5386.457} C_VEL
LIN {X 0,Y 501.437,Z 668.771,A -85,B 0,C 180,E1 5389.481,E2 5389.481} C_VEL
LIN {X 0,Y 500.236,Z 692.714,A -85,B 0,C 180,E1 5393.467,E2 5393.467} C_VEL
LIN {X 0,Y 499.744,Z 703.35,A -85,B 0,C 180,E1 5397.388,E2 5397.388} C_VEL
LIN {X 0,Y 499.91,Z 702.781,A -85,B 0,C 180,E1 5402.608,E2 5402.608} C_VEL
LIN {X 0,Y 500.486,Z 687.2,A -85,B 0,C 180,E1 5407.402,E2 5407.402} C_VEL
LIN {X 0,Y 501.547,Z 658.643,A -85,B 0,C 180,E1 5411.341,E2 5411.341} C_VEL
LIN {X 0,Y 502.653,Z 619.164,A -85,B 0,C 180,E1 5414.031,E2 5414.031} C_VEL
LIN {X 0,Y 499.261,Z 602.81,A -85,B 0,C 180,E1 5414.971,E2 5414.971} C_VEL
LIN {X 0,Y 498.611,Z 602.81,A -85,B 0,C 180,E1 5424.257,E2 5424.257} C_VEL
LIN {X 0,Y 498.128,Z 602.81,A -85,B 0,C 180,E1 5433.078,E2 5433.078} C_VEL
LIN {X 0,Y 498.14,Z 602.81,A -85,B 0,C 180,E1 5443.266,E2 5443.266} C_VEL
LIN {X 0,Y 498.004,Z 602.81,A -85,B 0,C 180,E1 5451.328,E2 5451.328} C_VEL
LIN {X 0,Y 498.241,Z 602.81,A -85,B 0,C 180,E1 5460.226,E2 5460.226} C_VEL
LIN {X 0,Y 498.022,Z 602.81,A -85,B 0,C 180,E1 5469.474,E2 5469.474} C_VEL
LIN {X 0,Y 498.47,Z 602.81,A -85,B 0,C 180,E1 5476.788,E2 5476.788} C_VEL
LIN {X 0,Y 498.801,Z 602.81,A -85,B 0,C 180,E1 5485.624,E2 5485.624} C_VEL
LIN {X 0,Y 498.839,Z 602.81,A -85,B 0,C 180,E1 5492.601,E2 5492.601} C_VEL
LIN {X 0,Y 498.789,Z 602.81,A -85,B 0,C 180,E1 5501.39,E2 5501.39} C_VEL
LIN {X 0,Y 498.699,Z 602.81,A -85,B 0,C 180,E1 5511.867,E2 5511.867} C_VEL
LIN {X 0,Y 498.408,Z 602.81,A -85,B 0,C 180,E1 5520.138,E2 5520.138} C_VEL
LIN {X 0,Y 498.316,Z 602.81,A -85,B 0,C 180,E1 5529.058,E2 5529.058} C_VEL
LIN {X 0,Y 498.17,Z 602.81,A -85,B 0,C 180,E1 5539.089,E2 5539.089} C_VEL
LIN {X 0,Y 498.11,Z 602.81,A -85,B 0,C 180,E1 5547.784,E2 5547.784} C_VEL
LIN {X 0,Y 498.408,Z 602.983,A -85,B 0,C 180,E1 5555.087,E2 5555.087} C_VEL
LIN {X 0,Y 506.857,Z 637.562,A -85,B 0,C 180,E1 5556.346,E2 5556.346} C_VEL
LIN {X 0,Y 504.394,Z 690.299,A -85,B 0,C 180,E1 5559.069,E2 5559.069} C_VEL
LIN {X 0,Y 502.015,Z 734.402,A -85,B 0,C 180,E1 5563.313,E2 5563.313} C_VEL
LIN {X 0,Y 500.191,Z 766.51,A -85,B 0,C 180,E1 5568.628,E2 5568.628} C_VEL
LIN {X 0,Y 499.277,Z 785.62,A -85,B 0,C 180,E1 5574.77,E2 5574.77} C_VEL
LIN {X 0,Y 498.932,Z 790.268,A -85,B 0,C 180,E1 5580.873,E2 5580.873} C_VEL
LIN {X 0,Y 499.28,Z 782.71,A -85,B 0,C 180,E1 5586.546,E2 5586.546} C_VEL
LIN {X 0,Y 500.187,Z 762.06,A -85,B 0,C 180,E1 5592.263,E2 5592.263} C_VEL
LIN {X 0,Y 502.201,Z 727.913,A -85,B 0,C 180,E1 5597.393,E2 5597.393} C_VEL
LIN {X 0,Y 504.826,Z 682.981,A -85,B 0,C 180,E1 5601.294,E2 5601.294} C_VEL
LIN {X 0,Y 506.449,Z 629.396,A -85,B 0,C 180,E1 5603.734,E2 5603.734} C_VEL
LIN {X 0,Y 498.463,Z 602.81,A -85,B 0,C 180,E1 5604.787,E2 5604.787} C_VEL
LIN {X 0,Y 498.293,Z 602.81,A -85,B 0,C 180,E1 5614.292,E2 5614.292} C_VEL
LIN {X 0,Y 498.26,Z 602.81,A -85,B 0,C 180,E1 5614.948,E2 5614.948} C_VEL
LIN {X 0,Y 490.206,Z 602.81,A -85,B 0,C 180,E1 5618.971,E2 5618.971} C_VEL
LIN {X 0,Y 490.112,Z 602.81,A -85,B 0,C 180,E1 5628.289,E2 5628.289} C_VEL
LIN {X 0,Y 490.149,Z 602.81,A -85,B 0,C 180,E1 5638.365,E2 5638.365} C_VEL
LIN {X 0,Y 490.812,Z 604.521,A -85,B 0,C 180,E1 5644.213,E2 5644.213} C_VEL
LIN {X 0,Y 499.287,Z 638.364,A -85,B 0,C 180,E1 5645.096,E2 5645.096} C_VEL
LIN {X 0,Y 498.188,Z 702.594,A -85,B 0,C 180,E1 5646.572,E2 5646.572} C_VEL
LIN {X 0,Y 495.844,Z 753.544,A -85,B 0,C 180,E1 5649.528,E2 5649.528} C_VEL
LIN {X 0,Y 493.579,Z 796.405,A -85,B 0,C 180,E1 5653.953,E2 5653.953} C_VEL
LIN {X 0,Y 492.206,Z 827.317,A -85,B 0,C 180,E1 5659.356,E2 5659.356} C_VEL
LIN {X 0,Y 491.412,Z 845.325,A -85,B 0,C 180,E1 5665.587,E2 5665.587} C_VEL
LIN {X 0,Y 491.341,Z 848.718,A -85,B 0,C 180,E1 5670.899,E2 5670.899} C_VEL
LIN {X 0,Y 491.263,Z 840.525,A -85,B 0,C 180,E1 5676.666,E2 5676.666} C_VEL
LIN {X 0,Y 491.969,Z 819.414,A -85,B 0,C 180,E1 5682.257,E2 5682.257} C_VEL
LIN {X 0,Y 493.775,Z 784.512,A -85,B 0,C 180,E1 5687.445,E2 5687.445} C_VEL
LIN {X 0,Y 496.513,Z 737.858,A -85,B 0,C 180,E1 5691.552,E2 5691.552} C_VEL
LIN {X 0,Y 498.812,Z 685.784,A -85,B 0,C 180,E1 5693.967,E2 5693.967} C_VEL
LIN {X 0,Y 497.369,Z 625.036,A -85,B 0,C 180,E1 5695.198,E2 5695.198} C_VEL
LIN {X 0,Y 490.708,Z 602.81,A -85,B 0,C 180,E1 5696.06,E2 5696.06} C_VEL
LIN {X 0,Y 490.334,Z 602.81,A -85,B 0,C 180,E1 5704.942,E2 5704.942} C_VEL
LIN {X 0,Y 490.294,Z 602.81,A -85,B 0,C 180,E1 5714.153,E2 5714.153} C_VEL
LIN {X 0,Y 490.181,Z 602.81,A -85,B 0,C 180,E1 5722.865,E2 5722.865} C_VEL
LIN {X 0,Y 490.251,Z 602.81,A -85,B 0,C 180,E1 5733.331,E2 5733.331} C_VEL
LIN {X 0,Y 490.367,Z 602.81,A -85,B 0,C 180,E1 5742.902,E2 5742.902} C_VEL
LIN {X 0,Y 490.711,Z 604.81,A -85,B 0,C 180,E1 5744.731,E2 5744.731} C_VEL
LIN {X 0,Y 495.064,Z 634.938,A -85,B 0,C 180,E1 5746.271,E2 5746.271} C_VEL
LIN {X 0,Y 493.671,Z 671.298,A -85,B 0,C 180,E1 5749.482,E2 5749.482} C_VEL
LIN {X 0,Y 492.486,Z 695.591,A -85,B 0,C 180,E1 5753.808,E2 5753.808} C_VEL
LIN {X 0,Y 491.868,Z 704.559,A -85,B 0,C 180,E1 5757.346,E2 5757.346} C_VEL
LIN {X 0,Y 492.015,Z 703.902,A -85,B 0,C 180,E1 5762.65,E2 5762.65} C_VEL
LIN {X 0,Y 492.633,Z 688.158,A -85,B 0,C 180,E1 5767.521,E2 5767.521} C_VEL
LIN {X 0,Y 493.774,Z 659.437,A -85,B 0,C 180,E1 5771.521,E2 5771.521} C_VEL
LIN {X 0,Y 494.85,Z 619.665,A -85,B 0,C 180,E1 5774.267,E2 5774.267} C_VEL
LIN {X 0,Y 491.196,Z 602.81,A -85,B 0,C 180,E1 5775.223,E2 5775.223} C_VEL
LIN {X 0,Y 490.537,Z 602.81,A -85,B 0,C 180,E1 5784.683,E2 5784.683} C_VEL
LIN {X 0,Y 490.038,Z 602.81,A -85,B 0,C 180,E1 5794.95,E2 5794.95} C_VEL
LIN {X 0,Y 490.139,Z 602.81,A -85,B 0,C 180,E1 5804.153,E2 5804.153} C_VEL
LIN {X 0,Y 489.985,Z 602.81,A -85,B 0,C 180,E1 5812.835,E2 5812.835} C_VEL
LIN {X 0,Y 490.282,Z 602.81,A -85,B 0,C 180,E1 5821.894,E2 5821.894} C_VEL
LIN {X 0,Y 490.598,Z 602.81,A -85,B 0,C 180,E1 5832.898,E2 5832.898} C_VEL
LIN {X 0,Y 491.082,Z 602.81,A -85,B 0,C 180,E1 5841.993,E2 5841.993} C_VEL
LIN {X 0,Y 490.991,Z 602.81,A -85,B 0,C 180,E1 5850.871,E2 5850.871} C_VEL
LIN {X 0,Y 490.686,Z 602.81,A -85,B 0,C 180,E1 5859.778,E2 5859.778} C_VEL
LIN {X 0,Y 490.604,Z 602.81,A -85,B 0,C 180,E1 5869.376,E2 5869.376} C_VEL
LIN {X 0,Y 490.492,Z 602.81,A -85,B 0,C 180,E1 5878.636,E2 5878.636} C_VEL
LIN {X 0,Y 490.294,Z 602.81,A -85,B 0,C 180,E1 5887.888,E2 5887.888} C_VEL
LIN {X 0,Y 490.22,Z 602.81,A -85,B 0,C 180,E1 5896.647,E2 5896.647} C_VEL
LIN {X 0,Y 490.134,Z 602.81,A -85,B 0,C 180,E1 5905.098,E2 5905.098} C_VEL
LIN {X 0,Y 490.57,Z 604.496,A -85,B 0,C 180,E1 5914.726,E2 5914.726} C_VEL
LIN {X 0,Y 499.391,Z 638.372,A -85,B 0,C 180,E1 5916.032,E2 5916.032} C_VEL
LIN {X 0,Y 496.8,Z 690.609,A -85,B 0,C 180,E1 5918.774,E2 5918.774} C_VEL
LIN {X 0,Y 494.254,Z 734.479,A -85,B 0,C 180,E1 5923.043,E2 5923.043} C_VEL
LIN {X 0,Y 492.308,Z 766.784,A -85,B 0,C 180,E1 5928.444,E2 5928.444} C_VEL
LIN {X 0,Y 491.322,Z 786.017,A -85,B 0,C 180,E1 5934.685,E2 5934.685} C_VEL
LIN {X 0,Y 490.979,Z 790.745,A -85,B 0,C 180,E1 5940.887,E2 5940.887} C_VEL
LIN {X 0,Y 491.405,Z 782.024,A -85,B 0,C 180,E1 5947.097,E2 5947.097} C_VEL
LIN {X 0,Y 492.558,Z 760.088,A -85,B 0,C 180,E1 5952.908,E2 5952.908} C_VEL
LIN {X 0,Y 494.728,Z 724.728,A -85,B 0,C 180,E1 5958.034,E2 5958.034} C_VEL
LIN {X 0,Y 497.489,Z 678.333,A -85,B 0,C 180,E1 5961.895,E2 5961.895} C_VEL
LIN {X 0,Y 497.585,Z 627.206,A -85,B 0,C 180,E1 5964.186,E2 5964.186} C_VEL
LIN {X 0,Y 490.472,Z 602.81,A -85,B 0,C 180,E1 5965.208,E2 5965.208} C_VEL
LIN {X 0,Y 490.271,Z 602.81,A -85,B 0,C 180,E1 5974.934,E2 5974.934} C_VEL
LIN {X 0,Y 490.206,Z 602.81,A -85,B 0,C 180,E1 5978.971,E2 5978.971} C_VEL
LIN {X 0,Y 482.17,Z 602.81,A -85,B 0,C 180,E1 5983.03,E2 5983.03} C_VEL
LIN {X 0,Y 482.126,Z 602.81,A -85,B 0,C 180,E1 5993.382,E2 5993.382} C_VEL
LIN {X 0,Y 482.674,Z 604.063,A -85,B 0,C 180,E1 6003.841,E2 6003.841} C_VEL
LIN {X 0,Y 491.791,Z 639.918,A -85,B 0,C 180,E1 6004.808,E2 6004.808} C_VEL
LIN {X 0,Y 490.596,Z 701.932,A -85,B 0,C 180,E1 6006.268,E2 6006.268} C_VEL
LIN {X 0,Y 488.03,Z 753.294,A -85,B 0,C 180,E1 6009.304,E2 6009.304} C_VEL
LIN {X 0,Y 485.615,Z 796.73,A -85,B 0,C 180,E1 6013.915,E2 6013.915} C_VEL
LIN {X 0,Y 484.128,Z 827.954,A -85,B 0,C 180,E1 6019.632,E2 6019.632} C_VEL
LIN {X 0,Y 483.509,Z 844.219,A -85,B 0,C 180,E1 6025.515,E2 6025.515} C_VEL
LIN {X 0,Y 483.419,Z 847.594,A -85,B 0,C 180,E1 6030.914,E2 6030.914} C_VEL
LIN {X 0,Y 483.346,Z 839.302,A -85,B 0,C 180,E1 6036.775,E2 6036.775} C_VEL
LIN {X 0,Y 484.074,Z 817.14,A -85,B 0,C 180,E1 6042.69,E2 6042.69} C_VEL
LIN {X 0,Y 486.073,Z 781.719,A -85,B 0,C 180,E1 6047.974,E2 6047.974} C_VEL
LIN {X 0,Y 489.041,Z 735.448,A -85,B 0,C 180,E1 6051.994,E2 6051.994} C_VEL
LIN {X 0,Y 491.49,Z 683.058,A -85,B 0,C 180,E1 6054.379,E2 6054.379} C_VEL
LIN {X 0,Y 489.719,Z 625.665,A -85,B 0,C 180,E1 6055.57,E2 6055.57} C_VEL
LIN {X 0,Y 482.663,Z 602.81,A -85,B 0,C 180,E1 6056.356,E2 6056.356} C_VEL
LIN {X 0,Y 482.25,Z 602.81,A -85,B 0,C 180,E1 6066.638,E2 6066.638} C_VEL
LIN {X 0,Y 482.231,Z 602.81,A -85,B 0,C 180,E1 6075.091,E2 6075.091} C_VEL
LIN {X 0,Y 482.087,Z 602.81,A -85,B 0,C 180,E1 6084.384,E2 6084.384} C_VEL
LIN {X 0,Y 482.209,Z 602.81,A -85,B 0,C 180,E1 6093.774,E2 6093.774} C_VEL
LIN {X 0,Y 482.381,Z 602.81,A -85,B 0,C 180,E1 6103.669,E2 6103.669} C_VEL
LIN {X 0,Y 482.876,Z 605.39,A -85,B 0,C 180,E1 6104.423,E2 6104.423} C_VEL
LIN {X 0,Y 487.487,Z 634.56,A -85,B 0,C 180,E1 6105.942,E2 6105.942} C_VEL
LIN {X 0,Y 485.93,Z 671.648,A -85,B 0,C 180,E1 6109.2,E2 6109.2} C_VEL
LIN {X 0,Y 484.532,Z 695.164,A -85,B 0,C 180,E1 6113.254,E2 6113.254} C_VEL
LIN {X 0,Y 483.984,Z 705.781,A -85,B 0,C 180,E1 6117.303,E2 6117.303} C_VEL
LIN {X 0,Y 484.104,Z 705.025,A -85,B 0,C 180,E1 6122.694,E2 6122.694} C_VEL
LIN {X 0,Y 484.792,Z 689.13,A -85,B 0,C 180,E1 6127.643,E2 6127.643} C_VEL
LIN {X 0,Y 485.995,Z 660.225,A -85,B 0,C 180,E1 6131.708,E2 6131.708} C_VEL
LIN {X 0,Y 486.937,Z 619.965,A -85,B 0,C 180,E1 6134.523,E2 6134.523} C_VEL
LIN {X 0,Y 483.119,Z 602.81,A -85,B 0,C 180,E1 6135.483,E2 6135.483} C_VEL
LIN {X 0,Y 482.36,Z 602.81,A -85,B 0,C 180,E1 6146.262,E2 6146.262} C_VEL
LIN {X 0,Y 481.962,Z 602.81,A -85,B 0,C 180,E1 6155.623,E2 6155.623} C_VEL
LIN {X 0,Y 482.135,Z 602.81,A -85,B 0,C 180,E1 6165.084,E2 6165.084} C_VEL
LIN {X 0,Y 482.024,Z 602.81,A -85,B 0,C 180,E1 6174.365,E2 6174.365} C_VEL
LIN {X 0,Y 482.262,Z 602.81,A -85,B 0,C 180,E1 6183.734,E2 6183.734} C_VEL
LIN {X 0,Y 482.594,Z 602.81,A -85,B 0,C 180,E1 6194.484,E2 6194.484} C_VEL
LIN {X 0,Y 482.915,Z 602.81,A -85,B 0,C 180,E1 6203.671,E2 6203.671} C_VEL
LIN {X 0,Y 482.986,Z 602.81,A -85,B 0,C 180,E1 6210.885,E2 6210.885} C_VEL
LIN {X 0,Y 482.689,Z 602.81,A -85,B 0,C 180,E1 6219.941,E2 6219.941} C_VEL
LIN {X 0,Y 482.615,Z 602.81,A -85,B 0,C 180,E1 6229.261,E2 6229.261} C_VEL
LIN {X 0,Y 482.382,Z 602.81,A -85,B 0,C 180,E1 6239.164,E2 6239.164} C_VEL
LIN {X 0,Y 482.259,Z 602.81,A -85,B 0,C 180,E1 6249.566,E2 6249.566} C_VEL
LIN {X 0,Y 482.151,Z 602.81,A -85,B 0,C 180,E1 6259.821,E2 6259.821} C_VEL
LIN {X 0,Y 482.189,Z 602.81,A -85,B 0,C 180,E1 6269.896,E2 6269.896} C_VEL
LIN {X 0,Y 482.553,Z 604.423,A -85,B 0,C 180,E1 6274.319,E2 6274.319} C_VEL
LIN {X 0,Y 491.918,Z 639.912,A -85,B 0,C 180,E1 6275.737,E2 6275.737} C_VEL
LIN {X 0,Y 489.098,Z 692.523,A -85,B 0,C 180,E1 6278.592,E2 6278.592} C_VEL
LIN {X 0,Y 486.368,Z 736.294,A -85,B 0,C 180,E1 6282.994,E2 6282.994} C_VEL
LIN {X 0,Y 484.453,Z 767.055,A -85,B 0,C 180,E1 6288.254,E2 6288.254} C_VEL
LIN {X 0,Y 483.388,Z 786.423,A -85,B 0,C 180,E1 6294.597,E2 6294.597} C_VEL
LIN {X 0,Y 482.994,Z 791.211,A -85,B 0,C 180,E1 6300.902,E2 6300.902} C_VEL
LIN {X 0,Y 483.454,Z 782.457,A -85,B 0,C 180,E1 6307.214,E2 6307.214} C_VEL
LIN {X 0,Y 484.861,Z 759.183,A -85,B 0,C 180,E1 6313.347,E2 6313.347} C_VEL
LIN {X 0,Y 487.228,Z 722.968,A -85,B 0,C 180,E1 6318.52,E2 6318.52} C_VEL
LIN {X 0,Y 490.013,Z 677.402,A -85,B 0,C 180,E1 6322.277,E2 6322.277} C_VEL
LIN {X 0,Y 489.939,Z 628.482,A -85,B 0,C 180,E1 6324.512,E2 6324.512} C_VEL
LIN {X 0,Y 482.441,Z 602.81,A -85,B 0,C 180,E1 6325.629,E2 6325.629} C_VEL
LIN {X 0,Y 482.196,Z 602.81,A -85,B 0,C 180,E1 6335.607,E2 6335.607} C_VEL
LIN {X 0,Y 482.17,Z 602.81,A -85,B 0,C 180,E1 6343.03,E2 6343.03} C_VEL
LIN {X 0,Y 473.963,Z 602.81,A -85,B 0,C 180,E1 6347.161,E2 6347.161} C_VEL
LIN {X 0,Y 474.021,Z 602.81,A -85,B 0,C 180,E1 6355.95,E2 6355.95} C_VEL
LIN {X 0,Y 474.655,Z 604.199,A -85,B 0,C 180,E1 6363.43,E2 6363.43} C_VEL
LIN {X 0,Y 484.28,Z 640.694,A -85,B 0,C 180,E1 6364.496,E2 6364.496} C_VEL
LIN {X 0,Y 482.985,Z 701.872,A -85,B 0,C 180,E1 6365.981,E2 6365.981} C_VEL
LIN {X 0,Y 480.222,Z 753.033,A -85,B 0,C 180,E1 6369.073,E2 6369.073} C_VEL
LIN {X 0,Y 477.723,Z 795.374,A -85,B 0,C 180,E1 6373.642,E2 6373.642} C_VEL
LIN {X 0,Y 476.206,Z 826.789,A -85,B 0,C 180,E1 6379.458,E2 6379.458} C_VEL
LIN {X 0,Y 475.616,Z 843.113,A -85,B 0,C 180,E1 6385.44,E2 6385.44} C_VEL
LIN {X 0,Y 475.507,Z 846.472,A -85,B 0,C 180,E1 6390.929,E2 6390.929} C_VEL
LIN {X 0,Y 475.371,Z 838.411,A -85,B 0,C 180,E1 6396.89,E2 6396.89} C_VEL
LIN {X 0,Y 476.14,Z 816.728,A -85,B 0,C 180,E1 6402.871,E2 6402.871} C_VEL
LIN {X 0,Y 478.258,Z 781.453,A -85,B 0,C 180,E1 6408.219,E2 6408.219} C_VEL
LIN {X 0,Y 481.456,Z 734.428,A -85,B 0,C 180,E1 6412.359,E2 6412.359} C_VEL
LIN {X 0,Y 484.113,Z 681.365,A -85,B 0,C 180,E1 6414.775,E2 6414.775} C_VEL
LIN {X 0,Y 482.442,Z 627.56,A -85,B 0,C 180,E1 6415.91,E2 6415.91} C_VEL
LIN {X 0,Y 474.624,Z 602.81,A -85,B 0,C 180,E1 6417.03,E2 6417.03} C_VEL
LIN {X 0,Y 474.234,Z 602.81,A -85,B 0,C 180,E1 6426.312,E2 6426.312} C_VEL
LIN {X 0,Y 474.105,Z 602.81,A -85,B 0,C 180,E1 6436.514,E2 6436.514} C_VEL
LIN {X 0,Y 474.044,Z 602.81,A -85,B 0,C 180,E1 6445.929,E2 6445.929} C_VEL
LIN {X 0,Y 474.18,Z 602.81,A -85,B 0,C 180,E1 6455.818,E2 6455.818} C_VEL
LIN {X 0,Y 474.495,Z 603.881,A -85,B 0,C 180,E1 6464.001,E2 6464.001} C_VEL
LIN {X 0,Y 479.822,Z 636.628,A -85,B 0,C 180,E1 6465.748,E2 6465.748} C_VEL
LIN {X 0,Y 478.195,Z 672.944,A -85,B 0,C 180,E1 6469.022,E2 6469.022} C_VEL
LIN {X 0,Y 476.704,Z 696.401,A -85,B 0,C 180,E1 6473.143,E2 6473.143} C_VEL
LIN {X 0,Y 476.089,Z 707.011,A -85,B 0,C 180,E1 6477.258,E2 6477.258} C_VEL
LIN {X 0,Y 476.203,Z 706.143,A -85,B 0,C 180,E1 6482.738,E2 6482.738} C_VEL
LIN {X 0,Y 476.932,Z 690.053,A -85,B 0,C 180,E1 6487.77,E2 6487.77} C_VEL
LIN {X 0,Y 478.222,Z 660.941,A -85,B 0,C 180,E1 6491.902,E2 6491.902} C_VEL
LIN {X 0,Y 479.063,Z 620.378,A -85,B 0,C 180,E1 6494.773,E2 6494.773} C_VEL
LIN {X 0,Y 475.088,Z 602.81,A -85,B 0,C 180,E1 6495.752,E2 6495.752} C_VEL
LIN {X 0,Y 474.39,Z 602.81,A -85,B 0,C 180,E1 6505.583,E2 6505.583} C_VEL
LIN {X 0,Y 473.932,Z 602.81,A -85,B 0,C 180,E1 6515.246,E2 6515.246} C_VEL
LIN {X 0,Y 474.031,Z 602.81,A -85,B 0,C 180,E1 6523.906,E2 6523.906} C_VEL
LIN {X 0,Y 473.977,Z 602.81,A -85,B 0,C 180,E1 6533.665,E2 6533.665} C_VEL
LIN {X 0,Y 474.193,Z 602.81,A -85,B 0,C 180,E1 6542.339,E2 6542.339} C_VEL
LIN {X 0,Y 474.438,Z 602.81,A -85,B 0,C 180,E1 6552.296,E2 6552.296} C_VEL
LIN {X 0,Y 475.041,Z 602.81,A -85,B 0,C 180,E1 6561.721,E2 6561.721} C_VEL
LIN {X 0,Y 474.997,Z 602.81,A -85,B 0,C 180,E1 6570.9,E2 6570.9} C_VEL
LIN {X 0,Y 474.679,Z 602.81,A -85,B 0,C 180,E1 6580.111,E2 6580.111} C_VEL
LIN {X 0,Y 474.593,Z 602.81,A -85,B 0,C 180,E1 6589.599,E2 6589.599} C_VEL
LIN {X 0,Y 474.332,Z 602.81,A -85,B 0,C 180,E1 6599.708,E2 6599.708} C_VEL
LIN {X 0,Y 474.254,Z 602.81,A -85,B 0,C 180,E1 6608.582,E2 6608.582} C_VEL
LIN {X 0,Y 474.067,Z 602.81,A -85,B 0,C 180,E1 6618.991,E2 6618.991} C_VEL
LIN {X 0,Y 474.045,Z 602.81,A -85,B 0,C 180,E1 6628.119,E2 6628.119} C_VEL
